REGION Network 72: CM Electrode Cutter Z Axis Command homing
   RUNG wire#powerrail
      Contact( #TRUE )
      Coil( "Unit1.Em4.ControlNodes".cm.Interlock.electrodeCutter.source.homing )
   END_RUNG
   RUNG wire#powerrail
      I_Contact( "Unit1.Em4.ControlNodes".cutter."step".action[113] )
      Not()
      Contact( "Unit1.Em4.ControlNodes".cm.Interlock.electrodeCutter.source.homing )
      Coil( "Unit1.Em4.ControlNodes".cmElectrodeCutterAxisZ.commands.homing )
   END_RUNG
   // the same network as SCL:
   "Unit1.Em4.ControlNodes".cm.Interlock.electrodeCutter.source.homing := #TRUE;
   "Unit1.Em4.ControlNodes".cmElectrodeCutterAxisZ.commands.homing := NOT (NOT "Unit1.Em4.ControlNodes".cutter."step".action[113]) AND "Unit1.Em4.ControlNodes".cm.Interlock.electrodeCutter.source.homing;
END_REGION

REGION Network 73: CM Electrode Cutter Z Axis Command posRelative
   RUNG wire#powerrail
      Contact( #TRUE )
      Coil( "Unit1.Em4.ControlNodes".cm.Interlock.electrodeCutter.source.posRelative )
   END_RUNG
   RUNG wire#powerrail
      I_Contact( "Unit1.Em4.ControlNodes".cutter."step".action[211] )
      Not()
      Coil( "Unit1.Em4.ControlNodes".cmElectrodeCutterAxisZ.commands.posRelative )
   END_RUNG
   // the same network as SCL:
   "Unit1.Em4.ControlNodes".cm.Interlock.electrodeCutter.source.posRelative := #TRUE;
   "Unit1.Em4.ControlNodes".cmElectrodeCutterAxisZ.commands.posRelative := NOT (NOT "Unit1.Em4.ControlNodes".cutter."step".action[211]);
END_REGION

REGION Network 74: CM Electrode Cutter Z Axis Command posAbsolute
   RUNG wire#powerrail
      Contact( #TRUE )
      Coil( "Unit1.Em4.ControlNodes".cm.Interlock.electrodeCutter.source.posAbsolute[0] )
   END_RUNG
   RUNG wire#powerrail
      I_Contact( "Unit1.Em4.ControlNodes".cutter."step".action[122] )
      Not()
      Coil( "Unit1.Em4.ControlNodes".cmElectrodeCutterAxisZ.commands.posAbsolute )
   END_RUNG
   // the same network as SCL:
   "Unit1.Em4.ControlNodes".cm.Interlock.electrodeCutter.source.posAbsolute[0] := #TRUE;
   "Unit1.Em4.ControlNodes".cmElectrodeCutterAxisZ.commands.posAbsolute := NOT (NOT "Unit1.Em4.ControlNodes".cutter."step".action[122]);
END_REGION

REGION Network 75: CM Electrode Cutter Z Axis Command gearInRelative
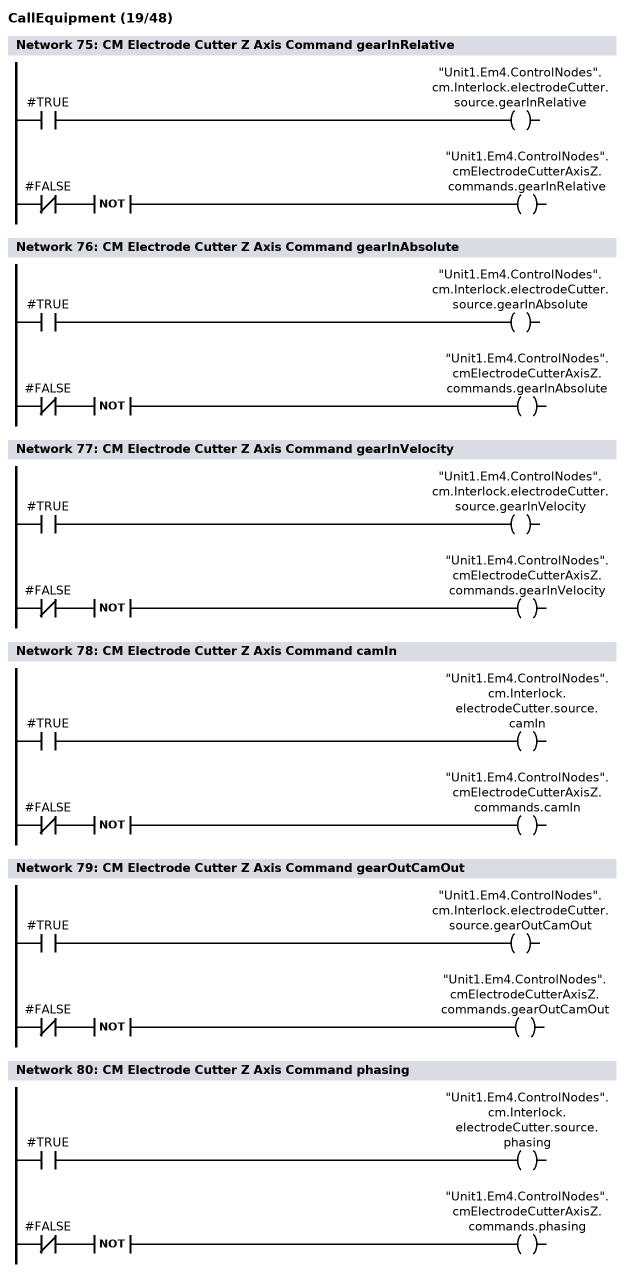
   RUNG wire#powerrail
      Contact( #TRUE )
      Coil( "Unit1.Em4.ControlNodes".cm.Interlock.electrodeCutter.source.gearInRelative )
   END_RUNG
   RUNG wire#powerrail
      I_Contact( #FALSE )
      Not()
      Coil( "Unit1.Em4.ControlNodes".cmElectrodeCutterAxisZ.commands.gearInRelative )
   END_RUNG
   // the same network as SCL:
   "Unit1.Em4.ControlNodes".cm.Interlock.electrodeCutter.source.gearInRelative := #TRUE;
   "Unit1.Em4.ControlNodes".cmElectrodeCutterAxisZ.commands.gearInRelative := NOT (NOT #FALSE);
END_REGION

REGION Network 76: CM Electrode Cutter Z Axis Command gearInAbsolute
   RUNG wire#powerrail
      Contact( #TRUE )
      Coil( "Unit1.Em4.ControlNodes".cm.Interlock.electrodeCutter.source.gearInAbsolute )
   END_RUNG
   RUNG wire#powerrail
      I_Contact( #FALSE )
      Not()
      Coil( "Unit1.Em4.ControlNodes".cmElectrodeCutterAxisZ.commands.gearInAbsolute )
   END_RUNG
   // the same network as SCL:
   "Unit1.Em4.ControlNodes".cm.Interlock.electrodeCutter.source.gearInAbsolute := #TRUE;
   "Unit1.Em4.ControlNodes".cmElectrodeCutterAxisZ.commands.gearInAbsolute := NOT (NOT #FALSE);
END_REGION

REGION Network 77: CM Electrode Cutter Z Axis Command gearInVelocity
   RUNG wire#powerrail
      Contact( #TRUE )
      Coil( "Unit1.Em4.ControlNodes".cm.Interlock.electrodeCutter.source.gearInVelocity )
   END_RUNG
   RUNG wire#powerrail
      I_Contact( #FALSE )
      Not()
      Coil( "Unit1.Em4.ControlNodes".cmElectrodeCutterAxisZ.commands.gearInVelocity )
   END_RUNG
   // the same network as SCL:
   "Unit1.Em4.ControlNodes".cm.Interlock.electrodeCutter.source.gearInVelocity := #TRUE;
   "Unit1.Em4.ControlNodes".cmElectrodeCutterAxisZ.commands.gearInVelocity := NOT (NOT #FALSE);
END_REGION

REGION Network 78: CM Electrode Cutter Z Axis Command camIn
   RUNG wire#powerrail
      Contact( #TRUE )
      Coil( "Unit1.Em4.ControlNodes".cm.Interlock.electrodeCutter.source.camIn )
   END_RUNG
   RUNG wire#powerrail
      I_Contact( #FALSE )
      Not()
      Coil( "Unit1.Em4.ControlNodes".cmElectrodeCutterAxisZ.commands.camIn )
   END_RUNG
   // the same network as SCL:
   "Unit1.Em4.ControlNodes".cm.Interlock.electrodeCutter.source.camIn := #TRUE;
   "Unit1.Em4.ControlNodes".cmElectrodeCutterAxisZ.commands.camIn := NOT (NOT #FALSE);
END_REGION

REGION Network 79: CM Electrode Cutter Z Axis Command gearOutCamOut
   RUNG wire#powerrail
      Contact( #TRUE )
      Coil( "Unit1.Em4.ControlNodes".cm.Interlock.electrodeCutter.source.gearOutCamOut )
   END_RUNG
   RUNG wire#powerrail
      I_Contact( #FALSE )
      Not()
      Coil( "Unit1.Em4.ControlNodes".cmElectrodeCutterAxisZ.commands.gearOutCamOut )
   END_RUNG
   // the same network as SCL:
   "Unit1.Em4.ControlNodes".cm.Interlock.electrodeCutter.source.gearOutCamOut := #TRUE;
   "Unit1.Em4.ControlNodes".cmElectrodeCutterAxisZ.commands.gearOutCamOut := NOT (NOT #FALSE);
END_REGION

REGION Network 80: CM Electrode Cutter Z Axis Command phasing
   RUNG wire#powerrail
      Contact( #TRUE )
      Coil( "Unit1.Em4.ControlNodes".cm.Interlock.electrodeCutter.source.phasing )
   END_RUNG
   RUNG wire#powerrail
      I_Contact( #FALSE )
      Not()
      Coil( "Unit1.Em4.ControlNodes".cmElectrodeCutterAxisZ.commands.phasing )
   END_RUNG
   // the same network as SCL:
   "Unit1.Em4.ControlNodes".cm.Interlock.electrodeCutter.source.phasing := #TRUE;
   "Unit1.Em4.ControlNodes".cmElectrodeCutterAxisZ.commands.phasing := NOT (NOT #FALSE);
END_REGION

REGION Network 81: CM Electrode Cutter Z Axis Command offset
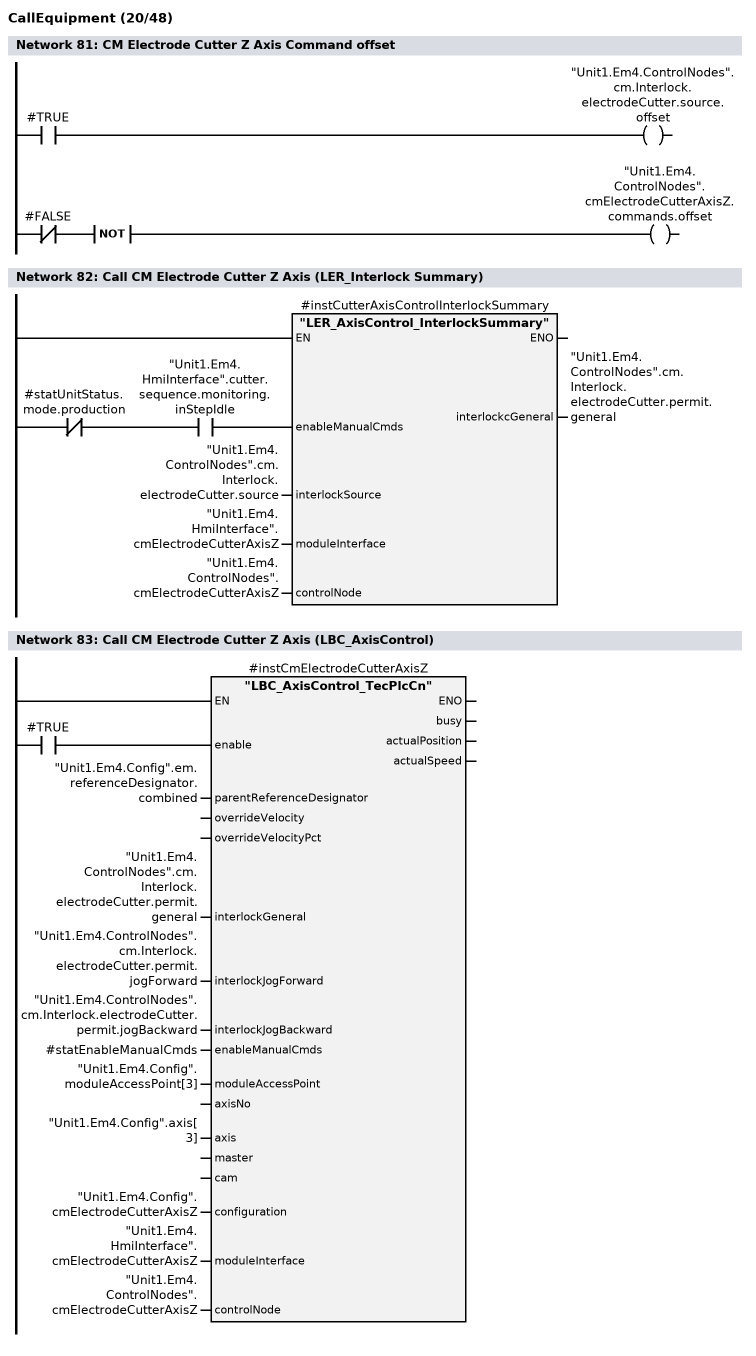
   RUNG wire#powerrail
      Contact( #TRUE )
      Coil( "Unit1.Em4.ControlNodes".cm.Interlock.electrodeCutter.source.offset )
   END_RUNG
   RUNG wire#powerrail
      I_Contact( #FALSE )
      Not()
      Coil( "Unit1.Em4.ControlNodes".cmElectrodeCutterAxisZ.commands.offset )
   END_RUNG
   // the same network as SCL:
   "Unit1.Em4.ControlNodes".cm.Interlock.electrodeCutter.source.offset := #TRUE;
   "Unit1.Em4.ControlNodes".cmElectrodeCutterAxisZ.commands.offset := NOT (NOT #FALSE);
END_REGION

REGION Network 82: Call CM Electrode Cutter Z Axis (LER_Interlock Summary)
   RUNG wire#powerrail
      #instCutterAxisControlInterlockSummary(enableManualCmds := wire#w1, interlockSource := "Unit1.Em4.ControlNodes".cm.Interlock.electrodeCutter.source, moduleInterface := "Unit1.Em4.HmiInterface".cmElectrodeCutterAxisZ, controlNode := "Unit1.Em4.ControlNodes".cmElectrodeCutterAxisZ, interlockcGeneral => "Unit1.Em4.ControlNodes".cm.Interlock.electrodeCutter.permit.general)
   END_RUNG
   RUNG wire#powerrail
      I_Contact( #statUnitStatus.mode.production )
      Contact( "Unit1.Em4.HmiInterface".cutter.sequence.monitoring.inStepIdle )
   END_RUNG wire#w1
   // the same network as SCL:
   #instCutterAxisControlInterlockSummary(enableManualCmds := NOT #statUnitStatus.mode.production AND "Unit1.Em4.HmiInterface".cutter.sequence.monitoring.inStepIdle,   // "LER_AxisControl_InterlockSummary"
                           interlockSource := "Unit1.Em4.ControlNodes".cm.Interlock.electrodeCutter.source,
                           moduleInterface := "Unit1.Em4.HmiInterface".cmElectrodeCutterAxisZ,
                           controlNode := "Unit1.Em4.ControlNodes".cmElectrodeCutterAxisZ,
                           interlockcGeneral => "Unit1.Em4.ControlNodes".cm.Interlock.electrodeCutter.permit.general);
END_REGION

REGION Network 83: Call CM Electrode Cutter Z Axis (LBC_AxisControl)
   RUNG wire#powerrail
      #instCmElectrodeCutterAxisZ(enable := wire#w1, parentReferenceDesignator := "Unit1.Em4.Config".em.referenceDesignator.combined, overrideVelocity :=, overrideVelocityPct :=, interlockGeneral := "Unit1.Em4.ControlNodes".cm.Interlock.electrodeCutter.permit.general, interlockJogForward := "Unit1.Em4.ControlNodes".cm.Interlock.electrodeCutter.permit.jogForward, interlockJogBackward := "Unit1.Em4.ControlNodes".cm.Interlock.electrodeCutter.permit.jogBackward, enableManualCmds := #statEnableManualCmds, moduleAccessPoint := "Unit1.Em4.Config".moduleAccessPoint[3], axisNo :=, axis := "Unit1.Em4.Config".axis[3], master :=, cam :=, configuration := "Unit1.Em4.Config".cmElectrodeCutterAxisZ, moduleInterface := "Unit1.Em4.HmiInterface".cmElectrodeCutterAxisZ, controlNode := "Unit1.Em4.ControlNodes".cmElectrodeCutterAxisZ, busy =>, actualPosition =>, actualSpeed =>)
   END_RUNG
   RUNG wire#powerrail
      Contact( #TRUE )
   END_RUNG wire#w1
   // the same network as SCL:
   #instCmElectrodeCutterAxisZ(enable := #TRUE,   // "LBC_AxisControl_TecPlcCn"
                           parentReferenceDesignator := "Unit1.Em4.Config".em.referenceDesignator.combined,
                           interlockGeneral := "Unit1.Em4.ControlNodes".cm.Interlock.electrodeCutter.permit.general,
                           interlockJogForward := "Unit1.Em4.ControlNodes".cm.Interlock.electrodeCutter.permit.jogForward,
                           interlockJogBackward := "Unit1.Em4.ControlNodes".cm.Interlock.electrodeCutter.permit.jogBackward,
                           enableManualCmds := #statEnableManualCmds,
                           moduleAccessPoint := "Unit1.Em4.Config".moduleAccessPoint[3],
                           axis := "Unit1.Em4.Config".axis[3],
                           configuration := "Unit1.Em4.Config".cmElectrodeCutterAxisZ,
                           moduleInterface := "Unit1.Em4.HmiInterface".cmElectrodeCutterAxisZ,
                           controlNode := "Unit1.Em4.ControlNodes".cmElectrodeCutterAxisZ);
END_REGION

REGION Network 84: Call CM Electrode Cutter Z Axis (LER_ServoTorqueCal)
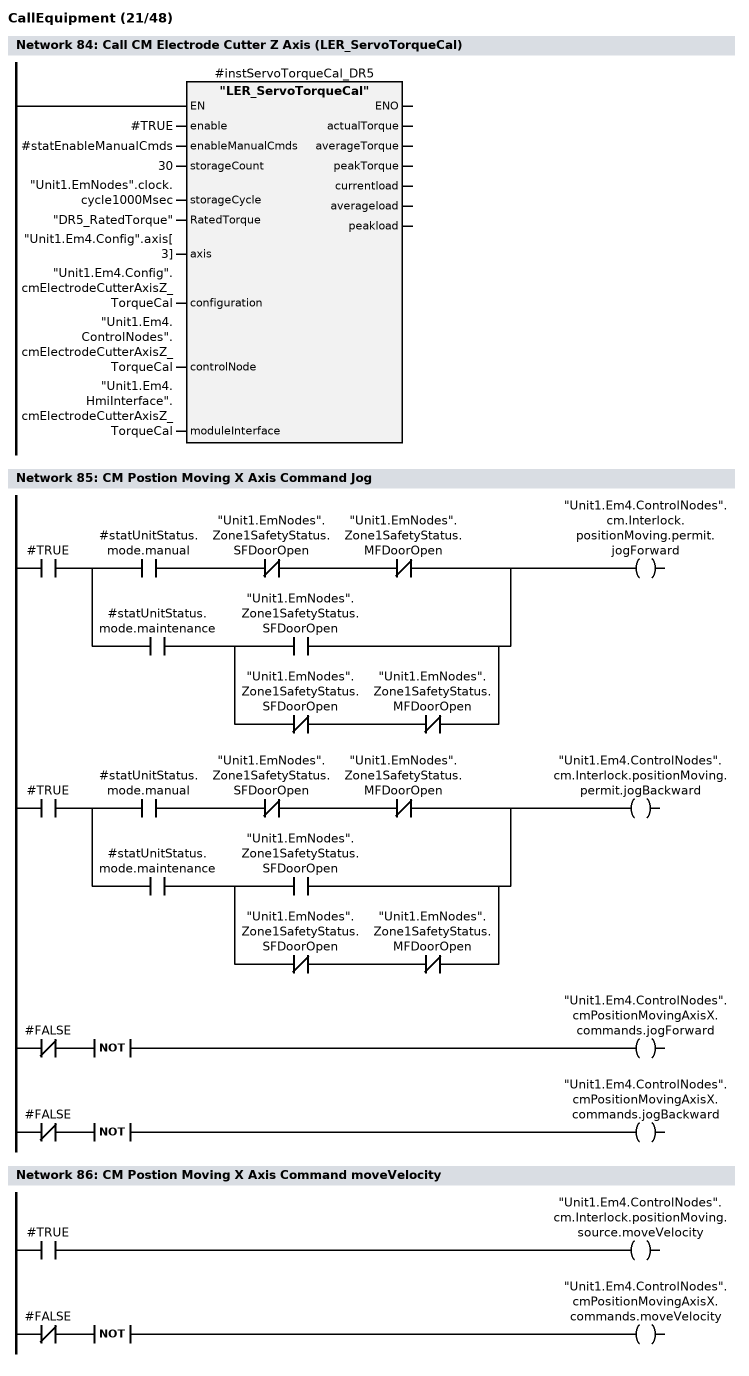
   RUNG wire#powerrail
      #instServoTorqueCal_DR5(enable := #TRUE, enableManualCmds := #statEnableManualCmds, storageCount := 30, storageCycle := "Unit1.EmNodes".clock.cycle1000Msec, RatedTorque := "DR5_RatedTorque", axis := "Unit1.Em4.Config".axis[3], configuration := "Unit1.Em4.Config".cmElectrodeCutterAxisZ_TorqueCal, controlNode := "Unit1.Em4.ControlNodes".cmElectrodeCutterAxisZ_TorqueCal, moduleInterface := "Unit1.Em4.HmiInterface".cmElectrodeCutterAxisZ_TorqueCal, actualTorque =>, averageTorque =>, peakTorque =>, currentload =>, averageload =>, peakload =>)
   END_RUNG
   // the same network as SCL:
   #instServoTorqueCal_DR5(enable := #TRUE,   // "LER_ServoTorqueCal"
                           enableManualCmds := #statEnableManualCmds,
                           storageCount := 30,
                           storageCycle := "Unit1.EmNodes".clock.cycle1000Msec,
                           RatedTorque := "DR5_RatedTorque",
                           axis := "Unit1.Em4.Config".axis[3],
                           configuration := "Unit1.Em4.Config".cmElectrodeCutterAxisZ_TorqueCal,
                           controlNode := "Unit1.Em4.ControlNodes".cmElectrodeCutterAxisZ_TorqueCal,
                           moduleInterface := "Unit1.Em4.HmiInterface".cmElectrodeCutterAxisZ_TorqueCal);
END_REGION

REGION Network 85: CM Postion Moving X Axis Command Jog
   RUNG wire#powerrail
      Contact( #TRUE )
      wire#w1
      Contact( #statUnitStatus.mode.manual )
      I_Contact( "Unit1.EmNodes".Zone1SafetyStatus.SFDoorOpen )
      I_Contact( "Unit1.EmNodes".Zone1SafetyStatus.MFDoorOpen )
      wire#w2
      Coil( "Unit1.Em4.ControlNodes".cm.Interlock.positionMoving.permit.jogForward )
   END_RUNG
   RUNG wire#w1
      Contact( #statUnitStatus.mode.maintenance )
      wire#w3
      Contact( "Unit1.EmNodes".Zone1SafetyStatus.SFDoorOpen )
   END_RUNG wire#w2
   RUNG wire#w3
      I_Contact( "Unit1.EmNodes".Zone1SafetyStatus.SFDoorOpen )
      I_Contact( "Unit1.EmNodes".Zone1SafetyStatus.MFDoorOpen )
   END_RUNG wire#w2
   RUNG wire#powerrail
      Contact( #TRUE )
      wire#w4
      Contact( #statUnitStatus.mode.manual )
      I_Contact( "Unit1.EmNodes".Zone1SafetyStatus.SFDoorOpen )
      I_Contact( "Unit1.EmNodes".Zone1SafetyStatus.MFDoorOpen )
      wire#w5
      Coil( "Unit1.Em4.ControlNodes".cm.Interlock.positionMoving.permit.jogBackward )
   END_RUNG
   RUNG wire#w4
      Contact( #statUnitStatus.mode.maintenance )
      wire#w6
      Contact( "Unit1.EmNodes".Zone1SafetyStatus.SFDoorOpen )
   END_RUNG wire#w5
   RUNG wire#w6
      I_Contact( "Unit1.EmNodes".Zone1SafetyStatus.SFDoorOpen )
      I_Contact( "Unit1.EmNodes".Zone1SafetyStatus.MFDoorOpen )
   END_RUNG wire#w5
   RUNG wire#powerrail
      I_Contact( #FALSE )
      Not()
      Coil( "Unit1.Em4.ControlNodes".cmPositionMovingAxisX.commands.jogForward )
   END_RUNG
   RUNG wire#powerrail
      I_Contact( #FALSE )
      Not()
      Coil( "Unit1.Em4.ControlNodes".cmPositionMovingAxisX.commands.jogBackward )
   END_RUNG
   // the same network as SCL:
   "Unit1.Em4.ControlNodes".cm.Interlock.positionMoving.permit.jogForward := #TRUE AND ((#statUnitStatus.mode.manual AND NOT "Unit1.EmNodes".Zone1SafetyStatus.SFDoorOpen AND NOT "Unit1.EmNodes".Zone1SafetyStatus.MFDoorOpen) OR (#statUnitStatus.mode.maintenance AND ("Unit1.EmNodes".Zone1SafetyStatus.SFDoorOpen OR (NOT "Unit1.EmNodes".Zone1SafetyStatus.SFDoorOpen AND NOT "Unit1.EmNodes".Zone1SafetyStatus.MFDoorOpen))));
   "Unit1.Em4.ControlNodes".cm.Interlock.positionMoving.permit.jogBackward := #TRUE AND ((#statUnitStatus.mode.manual AND NOT "Unit1.EmNodes".Zone1SafetyStatus.SFDoorOpen AND NOT "Unit1.EmNodes".Zone1SafetyStatus.MFDoorOpen) OR (#statUnitStatus.mode.maintenance AND ("Unit1.EmNodes".Zone1SafetyStatus.SFDoorOpen OR (NOT "Unit1.EmNodes".Zone1SafetyStatus.SFDoorOpen AND NOT "Unit1.EmNodes".Zone1SafetyStatus.MFDoorOpen))));
   "Unit1.Em4.ControlNodes".cmPositionMovingAxisX.commands.jogForward := NOT (NOT #FALSE);
   "Unit1.Em4.ControlNodes".cmPositionMovingAxisX.commands.jogBackward := NOT (NOT #FALSE);
END_REGION

REGION Network 86: CM Postion Moving X Axis Command moveVelocity
   RUNG wire#powerrail
      Contact( #TRUE )
      Coil( "Unit1.Em4.ControlNodes".cm.Interlock.positionMoving.source.moveVelocity )
   END_RUNG
   RUNG wire#powerrail
      I_Contact( #FALSE )
      Not()
      Coil( "Unit1.Em4.ControlNodes".cmPositionMovingAxisX.commands.moveVelocity )
   END_RUNG
   // the same network as SCL:
   "Unit1.Em4.ControlNodes".cm.Interlock.positionMoving.source.moveVelocity := #TRUE;
   "Unit1.Em4.ControlNodes".cmPositionMovingAxisX.commands.moveVelocity := NOT (NOT #FALSE);
END_REGION

REGION Network 87: CM Postion Moving X Axis Command stop
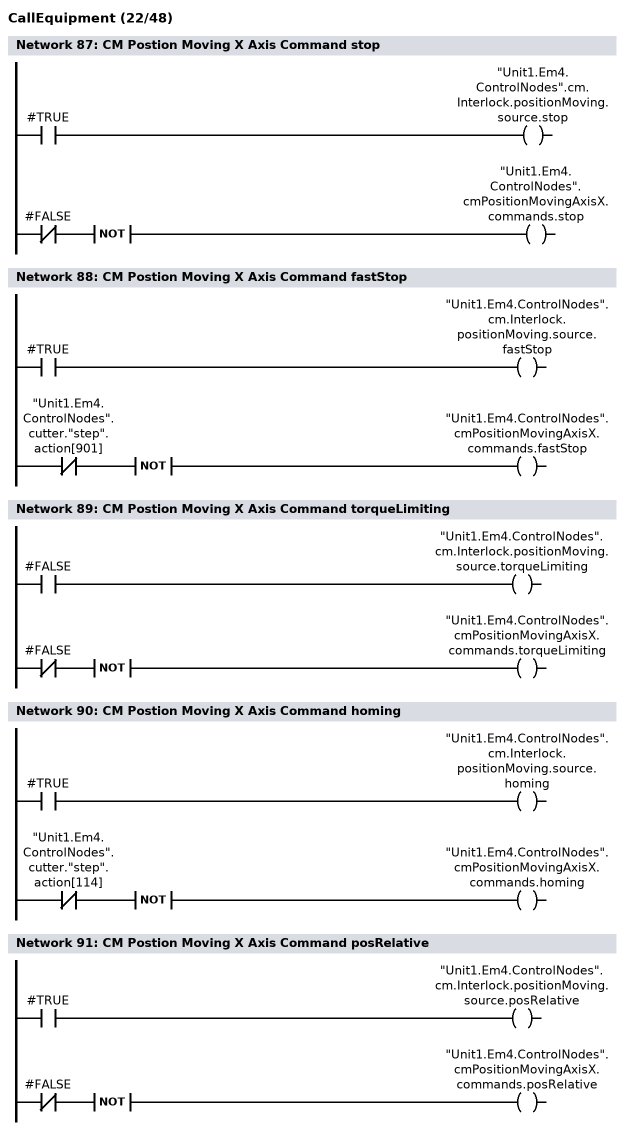
   RUNG wire#powerrail
      Contact( #TRUE )
      Coil( "Unit1.Em4.ControlNodes".cm.Interlock.positionMoving.source.stop )
   END_RUNG
   RUNG wire#powerrail
      I_Contact( #FALSE )
      Not()
      Coil( "Unit1.Em4.ControlNodes".cmPositionMovingAxisX.commands.stop )
   END_RUNG
   // the same network as SCL:
   "Unit1.Em4.ControlNodes".cm.Interlock.positionMoving.source.stop := #TRUE;
   "Unit1.Em4.ControlNodes".cmPositionMovingAxisX.commands.stop := NOT (NOT #FALSE);
END_REGION

REGION Network 88: CM Postion Moving X Axis Command fastStop
   RUNG wire#powerrail
      Contact( #TRUE )
      Coil( "Unit1.Em4.ControlNodes".cm.Interlock.positionMoving.source.fastStop )
   END_RUNG
   RUNG wire#powerrail
      I_Contact( "Unit1.Em4.ControlNodes".cutter."step".action[901] )
      Not()
      Coil( "Unit1.Em4.ControlNodes".cmPositionMovingAxisX.commands.fastStop )
   END_RUNG
   // the same network as SCL:
   "Unit1.Em4.ControlNodes".cm.Interlock.positionMoving.source.fastStop := #TRUE;
   "Unit1.Em4.ControlNodes".cmPositionMovingAxisX.commands.fastStop := NOT (NOT "Unit1.Em4.ControlNodes".cutter."step".action[901]);
END_REGION

REGION Network 89: CM Postion Moving X Axis Command torqueLimiting
   RUNG wire#powerrail
      Contact( #FALSE )
      Coil( "Unit1.Em4.ControlNodes".cm.Interlock.positionMoving.source.torqueLimiting )
   END_RUNG
   RUNG wire#powerrail
      I_Contact( #FALSE )
      Not()
      Coil( "Unit1.Em4.ControlNodes".cmPositionMovingAxisX.commands.torqueLimiting )
   END_RUNG
   // the same network as SCL:
   "Unit1.Em4.ControlNodes".cm.Interlock.positionMoving.source.torqueLimiting := #FALSE;
   "Unit1.Em4.ControlNodes".cmPositionMovingAxisX.commands.torqueLimiting := NOT (NOT #FALSE);
END_REGION

REGION Network 90: CM Postion Moving X Axis Command homing
   RUNG wire#powerrail
      Contact( #TRUE )
      Coil( "Unit1.Em4.ControlNodes".cm.Interlock.positionMoving.source.homing )
   END_RUNG
   RUNG wire#powerrail
      I_Contact( "Unit1.Em4.ControlNodes".cutter."step".action[114] )
      Not()
      Coil( "Unit1.Em4.ControlNodes".cmPositionMovingAxisX.commands.homing )
   END_RUNG
   // the same network as SCL:
   "Unit1.Em4.ControlNodes".cm.Interlock.positionMoving.source.homing := #TRUE;
   "Unit1.Em4.ControlNodes".cmPositionMovingAxisX.commands.homing := NOT (NOT "Unit1.Em4.ControlNodes".cutter."step".action[114]);
END_REGION

REGION Network 91: CM Postion Moving X Axis Command posRelative
   RUNG wire#powerrail
      Contact( #TRUE )
      Coil( "Unit1.Em4.ControlNodes".cm.Interlock.positionMoving.source.posRelative )
   END_RUNG
   RUNG wire#powerrail
      I_Contact( #FALSE )
      Not()
      Coil( "Unit1.Em4.ControlNodes".cmPositionMovingAxisX.commands.posRelative )
   END_RUNG
   // the same network as SCL:
   "Unit1.Em4.ControlNodes".cm.Interlock.positionMoving.source.posRelative := #TRUE;
   "Unit1.Em4.ControlNodes".cmPositionMovingAxisX.commands.posRelative := NOT (NOT #FALSE);
END_REGION

REGION Network 92: CM Postion Moving X Axis Command posAbsolute
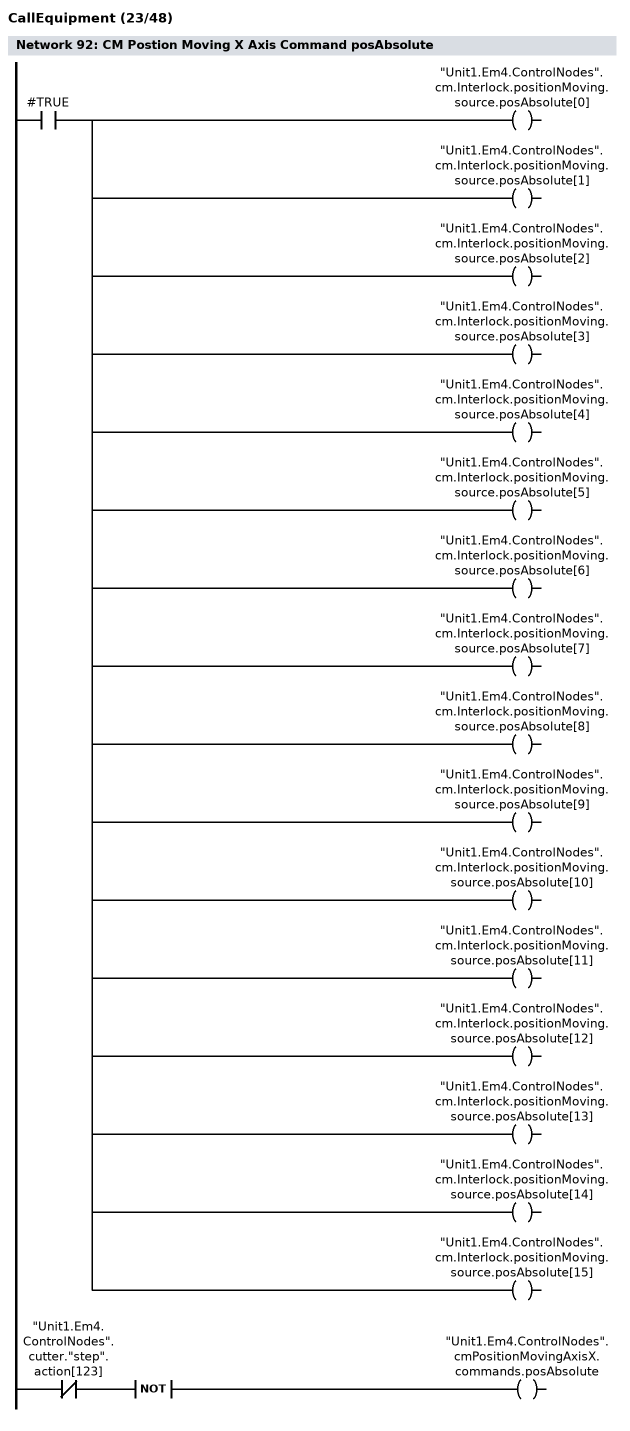
   RUNG wire#powerrail
      Contact( #TRUE )
      wire#w1
      Coil( "Unit1.Em4.ControlNodes".cm.Interlock.positionMoving.source.posAbsolute[0] )
   END_RUNG
   RUNG wire#w1
      Coil( "Unit1.Em4.ControlNodes".cm.Interlock.positionMoving.source.posAbsolute[1] )
   END_RUNG
   RUNG wire#w1
      Coil( "Unit1.Em4.ControlNodes".cm.Interlock.positionMoving.source.posAbsolute[2] )
   END_RUNG
   RUNG wire#w1
      Coil( "Unit1.Em4.ControlNodes".cm.Interlock.positionMoving.source.posAbsolute[3] )
   END_RUNG
   RUNG wire#w1
      Coil( "Unit1.Em4.ControlNodes".cm.Interlock.positionMoving.source.posAbsolute[4] )
   END_RUNG
   RUNG wire#w1
      Coil( "Unit1.Em4.ControlNodes".cm.Interlock.positionMoving.source.posAbsolute[5] )
   END_RUNG
   RUNG wire#w1
      Coil( "Unit1.Em4.ControlNodes".cm.Interlock.positionMoving.source.posAbsolute[6] )
   END_RUNG
   RUNG wire#w1
      Coil( "Unit1.Em4.ControlNodes".cm.Interlock.positionMoving.source.posAbsolute[7] )
   END_RUNG
   RUNG wire#w1
      Coil( "Unit1.Em4.ControlNodes".cm.Interlock.positionMoving.source.posAbsolute[8] )
   END_RUNG
   RUNG wire#w1
      Coil( "Unit1.Em4.ControlNodes".cm.Interlock.positionMoving.source.posAbsolute[9] )
   END_RUNG
   RUNG wire#w1
      Coil( "Unit1.Em4.ControlNodes".cm.Interlock.positionMoving.source.posAbsolute[10] )
   END_RUNG
   RUNG wire#w1
      Coil( "Unit1.Em4.ControlNodes".cm.Interlock.positionMoving.source.posAbsolute[11] )
   END_RUNG
   RUNG wire#w1
      Coil( "Unit1.Em4.ControlNodes".cm.Interlock.positionMoving.source.posAbsolute[12] )
   END_RUNG
   RUNG wire#w1
      Coil( "Unit1.Em4.ControlNodes".cm.Interlock.positionMoving.source.posAbsolute[13] )
   END_RUNG
   RUNG wire#w1
      Coil( "Unit1.Em4.ControlNodes".cm.Interlock.positionMoving.source.posAbsolute[14] )
   END_RUNG
   RUNG wire#w1
      Coil( "Unit1.Em4.ControlNodes".cm.Interlock.positionMoving.source.posAbsolute[15] )
   END_RUNG
   RUNG wire#powerrail
      I_Contact( "Unit1.Em4.ControlNodes".cutter."step".action[123] )
      Not()
      Coil( "Unit1.Em4.ControlNodes".cmPositionMovingAxisX.commands.posAbsolute )
   END_RUNG
   // the same network as SCL:
   "Unit1.Em4.ControlNodes".cm.Interlock.positionMoving.source.posAbsolute[0] := #TRUE;
   "Unit1.Em4.ControlNodes".cm.Interlock.positionMoving.source.posAbsolute[1] := #TRUE;
   "Unit1.Em4.ControlNodes".cm.Interlock.positionMoving.source.posAbsolute[2] := #TRUE;
   "Unit1.Em4.ControlNodes".cm.Interlock.positionMoving.source.posAbsolute[3] := #TRUE;
   "Unit1.Em4.ControlNodes".cm.Interlock.positionMoving.source.posAbsolute[4] := #TRUE;
   "Unit1.Em4.ControlNodes".cm.Interlock.positionMoving.source.posAbsolute[5] := #TRUE;
   "Unit1.Em4.ControlNodes".cm.Interlock.positionMoving.source.posAbsolute[6] := #TRUE;
   "Unit1.Em4.ControlNodes".cm.Interlock.positionMoving.source.posAbsolute[7] := #TRUE;
   "Unit1.Em4.ControlNodes".cm.Interlock.positionMoving.source.posAbsolute[8] := #TRUE;
   "Unit1.Em4.ControlNodes".cm.Interlock.positionMoving.source.posAbsolute[9] := #TRUE;
   "Unit1.Em4.ControlNodes".cm.Interlock.positionMoving.source.posAbsolute[10] := #TRUE;
   "Unit1.Em4.ControlNodes".cm.Interlock.positionMoving.source.posAbsolute[11] := #TRUE;
   "Unit1.Em4.ControlNodes".cm.Interlock.positionMoving.source.posAbsolute[12] := #TRUE;
   "Unit1.Em4.ControlNodes".cm.Interlock.positionMoving.source.posAbsolute[13] := #TRUE;
   "Unit1.Em4.ControlNodes".cm.Interlock.positionMoving.source.posAbsolute[14] := #TRUE;
   "Unit1.Em4.ControlNodes".cm.Interlock.positionMoving.source.posAbsolute[15] := #TRUE;
   "Unit1.Em4.ControlNodes".cmPositionMovingAxisX.commands.posAbsolute := NOT (NOT "Unit1.Em4.ControlNodes".cutter."step".action[123]);
END_REGION

REGION Network 93: Call CM Postion Moving X Axis (LER_Interlock Summary)
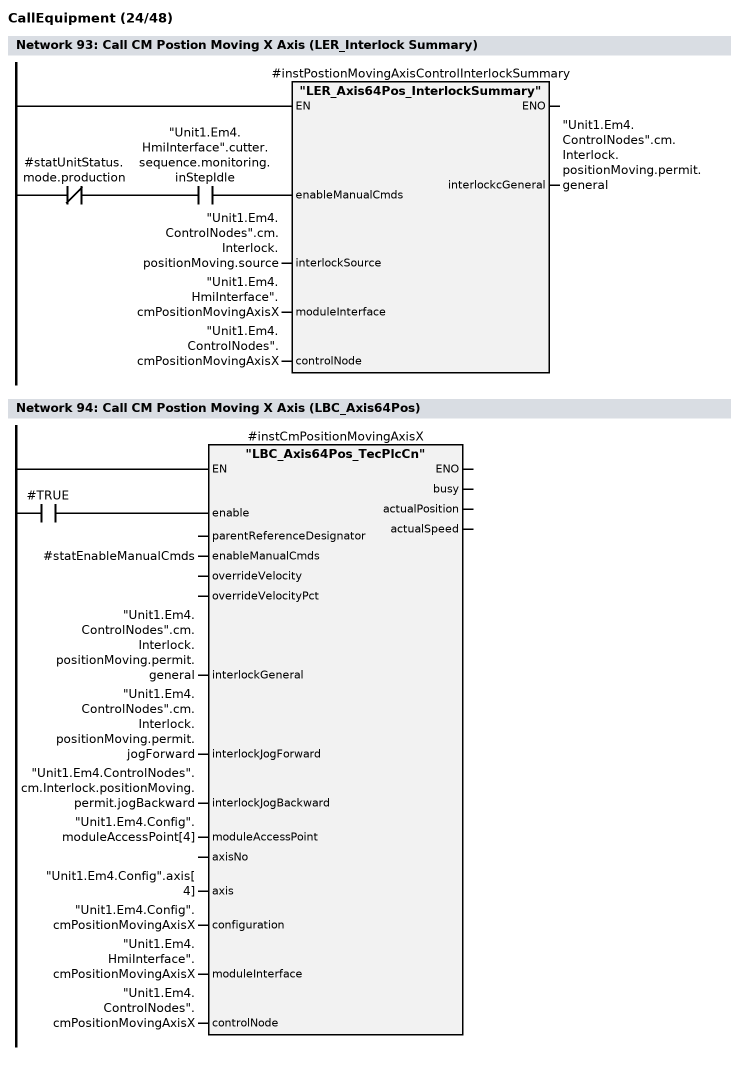
   RUNG wire#powerrail
      #instPostionMovingAxisControlInterlockSummary(enableManualCmds := wire#w1, interlockSource := "Unit1.Em4.ControlNodes".cm.Interlock.positionMoving.source, moduleInterface := "Unit1.Em4.HmiInterface".cmPositionMovingAxisX, controlNode := "Unit1.Em4.ControlNodes".cmPositionMovingAxisX, interlockcGeneral => "Unit1.Em4.ControlNodes".cm.Interlock.positionMoving.permit.general)
   END_RUNG
   RUNG wire#powerrail
      I_Contact( #statUnitStatus.mode.production )
      Contact( "Unit1.Em4.HmiInterface".cutter.sequence.monitoring.inStepIdle )
   END_RUNG wire#w1
   // the same network as SCL:
   #instPostionMovingAxisControlInterlockSummary(enableManualCmds := NOT #statUnitStatus.mode.production AND "Unit1.Em4.HmiInterface".cutter.sequence.monitoring.inStepIdle,   // "LER_Axis64Pos_InterlockSummary"
                           interlockSource := "Unit1.Em4.ControlNodes".cm.Interlock.positionMoving.source,
                           moduleInterface := "Unit1.Em4.HmiInterface".cmPositionMovingAxisX,
                           controlNode := "Unit1.Em4.ControlNodes".cmPositionMovingAxisX,
                           interlockcGeneral => "Unit1.Em4.ControlNodes".cm.Interlock.positionMoving.permit.general);
END_REGION

REGION Network 94: Call CM Postion Moving X Axis (LBC_Axis64Pos)
   RUNG wire#powerrail
      #instCmPositionMovingAxisX(enable := wire#w1, parentReferenceDesignator :=, enableManualCmds := #statEnableManualCmds, overrideVelocity :=, overrideVelocityPct :=, interlockGeneral := "Unit1.Em4.ControlNodes".cm.Interlock.positionMoving.permit.general, interlockJogForward := "Unit1.Em4.ControlNodes".cm.Interlock.positionMoving.permit.jogForward, interlockJogBackward := "Unit1.Em4.ControlNodes".cm.Interlock.positionMoving.permit.jogBackward, moduleAccessPoint := "Unit1.Em4.Config".moduleAccessPoint[4], axisNo :=, axis := "Unit1.Em4.Config".axis[4], configuration := "Unit1.Em4.Config".cmPositionMovingAxisX, moduleInterface := "Unit1.Em4.HmiInterface".cmPositionMovingAxisX, controlNode := "Unit1.Em4.ControlNodes".cmPositionMovingAxisX, busy =>, actualPosition =>, actualSpeed =>)
   END_RUNG
   RUNG wire#powerrail
      Contact( #TRUE )
   END_RUNG wire#w1
   // the same network as SCL:
   #instCmPositionMovingAxisX(enable := #TRUE,   // "LBC_Axis64Pos_TecPlcCn"
                           enableManualCmds := #statEnableManualCmds,
                           interlockGeneral := "Unit1.Em4.ControlNodes".cm.Interlock.positionMoving.permit.general,
                           interlockJogForward := "Unit1.Em4.ControlNodes".cm.Interlock.positionMoving.permit.jogForward,
                           interlockJogBackward := "Unit1.Em4.ControlNodes".cm.Interlock.positionMoving.permit.jogBackward,
                           moduleAccessPoint := "Unit1.Em4.Config".moduleAccessPoint[4],
                           axis := "Unit1.Em4.Config".axis[4],
                           configuration := "Unit1.Em4.Config".cmPositionMovingAxisX,
                           moduleInterface := "Unit1.Em4.HmiInterface".cmPositionMovingAxisX,
                           controlNode := "Unit1.Em4.ControlNodes".cmPositionMovingAxisX);
END_REGION

REGION Network 95: Call CM Postion Moving X Axis (LER_ServoTorqueCal)
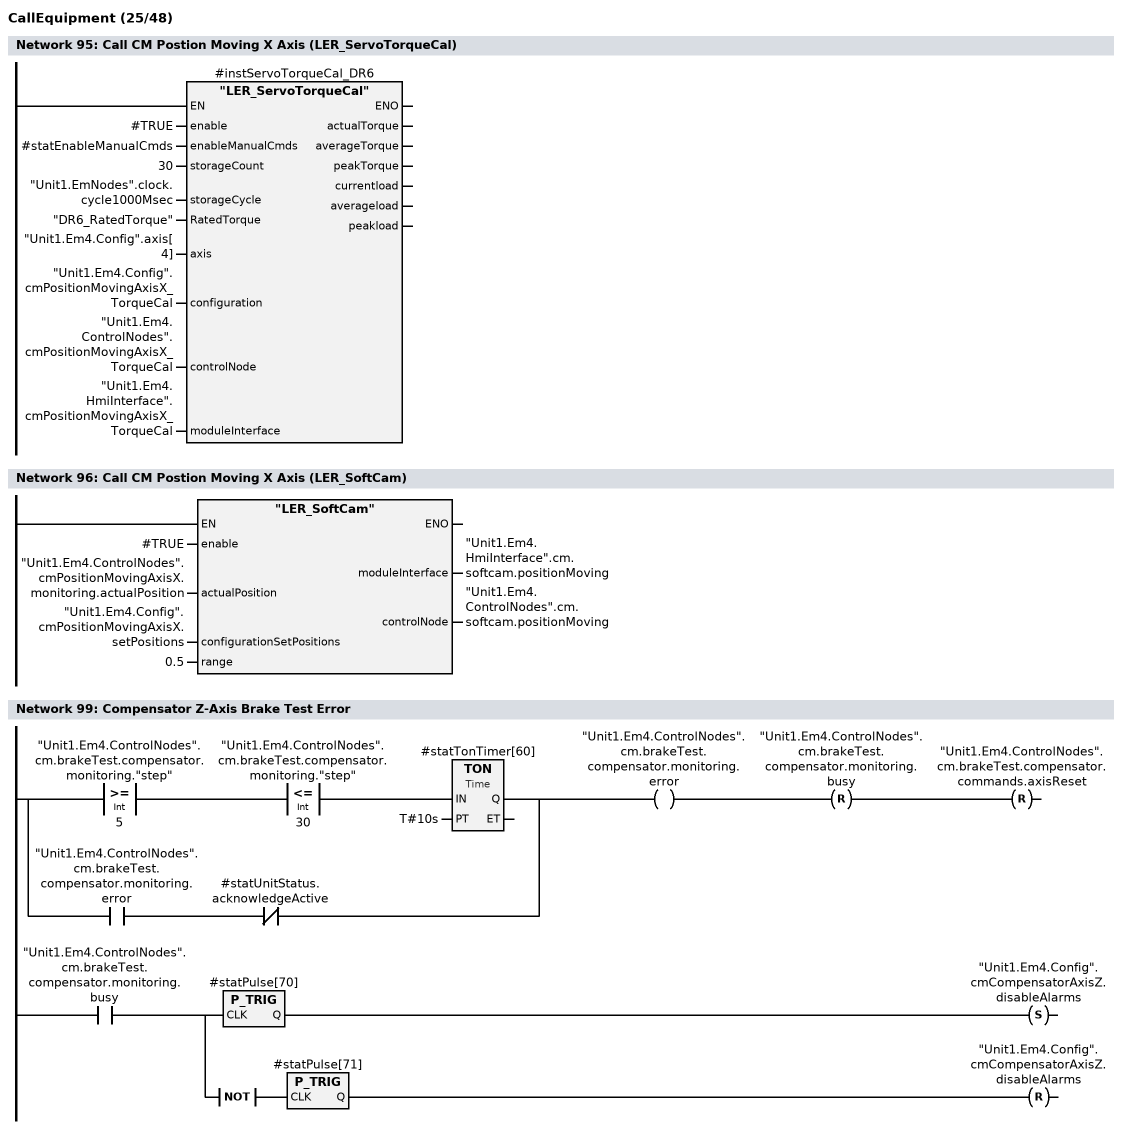
   RUNG wire#powerrail
      #instServoTorqueCal_DR6(enable := #TRUE, enableManualCmds := #statEnableManualCmds, storageCount := 30, storageCycle := "Unit1.EmNodes".clock.cycle1000Msec, RatedTorque := "DR6_RatedTorque", axis := "Unit1.Em4.Config".axis[4], configuration := "Unit1.Em4.Config".cmPositionMovingAxisX_TorqueCal, controlNode := "Unit1.Em4.ControlNodes".cmPositionMovingAxisX_TorqueCal, moduleInterface := "Unit1.Em4.HmiInterface".cmPositionMovingAxisX_TorqueCal, actualTorque =>, averageTorque =>, peakTorque =>, currentload =>, averageload =>, peakload =>)
   END_RUNG
   // the same network as SCL:
   #instServoTorqueCal_DR6(enable := #TRUE,   // "LER_ServoTorqueCal"
                           enableManualCmds := #statEnableManualCmds,
                           storageCount := 30,
                           storageCycle := "Unit1.EmNodes".clock.cycle1000Msec,
                           RatedTorque := "DR6_RatedTorque",
                           axis := "Unit1.Em4.Config".axis[4],
                           configuration := "Unit1.Em4.Config".cmPositionMovingAxisX_TorqueCal,
                           controlNode := "Unit1.Em4.ControlNodes".cmPositionMovingAxisX_TorqueCal,
                           moduleInterface := "Unit1.Em4.HmiInterface".cmPositionMovingAxisX_TorqueCal);
END_REGION

REGION Network 96: Call CM Postion Moving X Axis (LER_SoftCam)
   RUNG wire#powerrail
      "LER_SoftCam"(enable := #TRUE, actualPosition := "Unit1.Em4.ControlNodes".cmPositionMovingAxisX.monitoring.actualPosition, configurationSetPositions := "Unit1.Em4.Config".cmPositionMovingAxisX.setPositions, range := 0.5, moduleInterface => "Unit1.Em4.HmiInterface".cm.softcam.positionMoving, controlNode => "Unit1.Em4.ControlNodes".cm.softcam.positionMoving)
   END_RUNG
   // the same network as SCL:
   "LER_SoftCam"(enable := #TRUE,
                 actualPosition := "Unit1.Em4.ControlNodes".cmPositionMovingAxisX.monitoring.actualPosition,
                 configurationSetPositions := "Unit1.Em4.Config".cmPositionMovingAxisX.setPositions,
                 range := 0.5,
                 moduleInterface => "Unit1.Em4.HmiInterface".cm.softcam.positionMoving,
                 controlNode => "Unit1.Em4.ControlNodes".cm.softcam.positionMoving);
END_REGION

REGION Network 98: ******************** Brake Test (Axis) ********************
END_REGION

REGION Network 99: Compensator Z-Axis Brake Test Error
   RUNG wire#powerrail
      { S7_Templates := "SrcType := Int" } GE_Contact(in1 := "Unit1.Em4.ControlNodes".cm.brakeTest.compensator.monitoring."step", in2 := 5)
      { S7_Templates := "SrcType := Int" } LE_Contact(in1 := "Unit1.Em4.ControlNodes".cm.brakeTest.compensator.monitoring."step", in2 := 30)
      { S7_Templates := "time_type := Time" } #statTonTimer[60].TON(pt := T#10s, et =>)
      wire#w1
      Coil( "Unit1.Em4.ControlNodes".cm.brakeTest.compensator.monitoring.error )
      R_Coil( "Unit1.Em4.ControlNodes".cm.brakeTest.compensator.monitoring.busy )
      R_Coil( "Unit1.Em4.ControlNodes".cm.brakeTest.compensator.commands.axisReset )
   END_RUNG
   RUNG wire#powerrail
      Contact( "Unit1.Em4.ControlNodes".cm.brakeTest.compensator.monitoring.error )
      I_Contact( #statUnitStatus.acknowledgeActive )
   END_RUNG wire#w1
   RUNG wire#powerrail
      Contact( "Unit1.Em4.ControlNodes".cm.brakeTest.compensator.monitoring.busy )
      wire#w2
      P_Trig( #statPulse[70] )
      S_Coil( "Unit1.Em4.Config".cmCompensatorAxisZ.disableAlarms )
   END_RUNG
   RUNG wire#w2
      Not()
      P_Trig( #statPulse[71] )
      R_Coil( "Unit1.Em4.Config".cmCompensatorAxisZ.disableAlarms )
   END_RUNG
   // the same network as SCL:
   #statTonTimer[60].TON(IN := ("Unit1.Em4.ControlNodes".cm.brakeTest.compensator.monitoring."step" >= 5) AND ("Unit1.Em4.ControlNodes".cm.brakeTest.compensator.monitoring."step" <= 30),
                         PT := T#10s);
   "Unit1.Em4.ControlNodes".cm.brakeTest.compensator.monitoring.error := #statTonTimer[60].Q OR ("Unit1.Em4.ControlNodes".cm.brakeTest.compensator.monitoring.error AND NOT #statUnitStatus.acknowledgeActive);
   IF "Unit1.Em4.ControlNodes".cm.brakeTest.compensator.monitoring.error THEN
       "Unit1.Em4.ControlNodes".cm.brakeTest.compensator.monitoring.busy := FALSE;
       "Unit1.Em4.ControlNodes".cm.brakeTest.compensator.commands.axisReset := FALSE;
   END_IF;
   #_w1 := "Unit1.Em4.ControlNodes".cm.brakeTest.compensator.monitoring.busy AND NOT #statPulse[70];   // rising edge
   #statPulse[70] := "Unit1.Em4.ControlNodes".cm.brakeTest.compensator.monitoring.busy;
   IF #_w1 THEN "Unit1.Em4.Config".cmCompensatorAxisZ.disableAlarms := TRUE; END_IF;
   #_w2 := NOT "Unit1.Em4.ControlNodes".cm.brakeTest.compensator.monitoring.busy AND NOT #statPulse[71];   // rising edge
   #statPulse[71] := NOT "Unit1.Em4.ControlNodes".cm.brakeTest.compensator.monitoring.busy;
   IF #_w2 THEN "Unit1.Em4.Config".cmCompensatorAxisZ.disableAlarms := FALSE; END_IF;
END_REGION

REGION Network 100: Compensator Z-Axis Brake Test Initialize
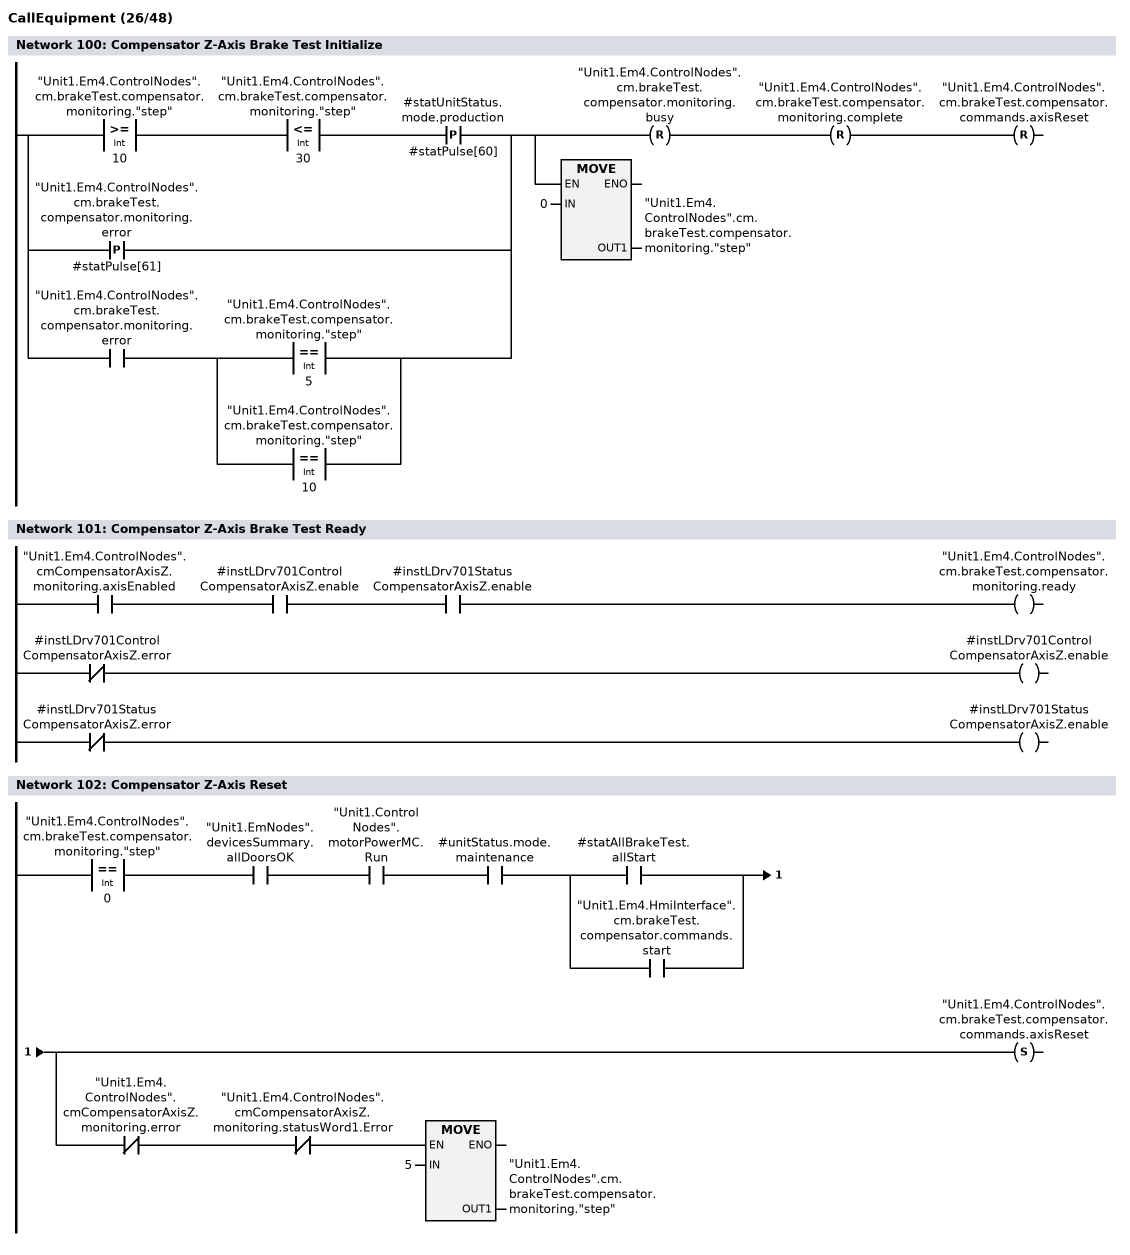
   RUNG wire#powerrail
      { S7_Templates := "SrcType := Int" } GE_Contact(in1 := "Unit1.Em4.ControlNodes".cm.brakeTest.compensator.monitoring."step", in2 := 10)
      { S7_Templates := "SrcType := Int" } LE_Contact(in1 := "Unit1.Em4.ControlNodes".cm.brakeTest.compensator.monitoring."step", in2 := 30)
      P_Contact(operand := #statUnitStatus.mode.production, bit := #statPulse[60])
      wire#w1
      R_Coil( "Unit1.Em4.ControlNodes".cm.brakeTest.compensator.monitoring.busy )
      R_Coil( "Unit1.Em4.ControlNodes".cm.brakeTest.compensator.monitoring.complete )
      R_Coil( "Unit1.Em4.ControlNodes".cm.brakeTest.compensator.commands.axisReset )
   END_RUNG
   RUNG wire#powerrail
      P_Contact(operand := "Unit1.Em4.ControlNodes".cm.brakeTest.compensator.monitoring.error, bit := #statPulse[61])
   END_RUNG wire#w1
   RUNG wire#powerrail
      Contact( "Unit1.Em4.ControlNodes".cm.brakeTest.compensator.monitoring.error )
      wire#w2
      { S7_Templates := "SrcType := Int" } EQ_Contact(in1 := "Unit1.Em4.ControlNodes".cm.brakeTest.compensator.monitoring."step", in2 := 5)
   END_RUNG wire#w1
   RUNG wire#w2
      { S7_Templates := "SrcType := Int" } EQ_Contact(in1 := "Unit1.Em4.ControlNodes".cm.brakeTest.compensator.monitoring."step", in2 := 10)
   END_RUNG wire#w1
   RUNG wire#w1
      Move(in := 0, out1 => "Unit1.Em4.ControlNodes".cm.brakeTest.compensator.monitoring."step")
   END_RUNG
   // the same network as SCL:
   #_w1 := ("Unit1.Em4.ControlNodes".cm.brakeTest.compensator.monitoring."step" >= 10) AND ("Unit1.Em4.ControlNodes".cm.brakeTest.compensator.monitoring."step" <= 30) AND #statUnitStatus.mode.production AND NOT #statPulse[60];   // rising edge of #statUnitStatus.mode.production
   #statPulse[60] := #statUnitStatus.mode.production;
   #_w2 := "Unit1.Em4.ControlNodes".cm.brakeTest.compensator.monitoring.error AND NOT #statPulse[61];   // rising edge of "Unit1.Em4.ControlNodes".cm.brakeTest.compensator.monitoring.error
   #statPulse[61] := "Unit1.Em4.ControlNodes".cm.brakeTest.compensator.monitoring.error;
   IF #_w1 OR #_w2 OR ("Unit1.Em4.ControlNodes".cm.brakeTest.compensator.monitoring.error AND (("Unit1.Em4.ControlNodes".cm.brakeTest.compensator.monitoring."step" = 5) OR ("Unit1.Em4.ControlNodes".cm.brakeTest.compensator.monitoring."step" = 10))) THEN
       "Unit1.Em4.ControlNodes".cm.brakeTest.compensator.monitoring.busy := FALSE;
       "Unit1.Em4.ControlNodes".cm.brakeTest.compensator.monitoring.complete := FALSE;
       "Unit1.Em4.ControlNodes".cm.brakeTest.compensator.commands.axisReset := FALSE;
       "Unit1.Em4.ControlNodes".cm.brakeTest.compensator.monitoring."step" := 0;
   END_IF;
END_REGION

REGION Network 101: Compensator Z-Axis Brake Test Ready
   RUNG wire#powerrail
      Contact( "Unit1.Em4.ControlNodes".cmCompensatorAxisZ.monitoring.axisEnabled )
      Contact( #instLDrv701ControlCompensatorAxisZ.enable )
      Contact( #instLDrv701StatusCompensatorAxisZ.enable )
      Coil( "Unit1.Em4.ControlNodes".cm.brakeTest.compensator.monitoring.ready )
   END_RUNG
   RUNG wire#powerrail
      I_Contact( #instLDrv701ControlCompensatorAxisZ.error )
      Coil( #instLDrv701ControlCompensatorAxisZ.enable )
   END_RUNG
   RUNG wire#powerrail
      I_Contact( #instLDrv701StatusCompensatorAxisZ.error )
      Coil( #instLDrv701StatusCompensatorAxisZ.enable )
   END_RUNG
   // the same network as SCL:
   "Unit1.Em4.ControlNodes".cm.brakeTest.compensator.monitoring.ready := "Unit1.Em4.ControlNodes".cmCompensatorAxisZ.monitoring.axisEnabled AND #instLDrv701ControlCompensatorAxisZ.enable AND #instLDrv701StatusCompensatorAxisZ.enable;
   #instLDrv701ControlCompensatorAxisZ.enable := NOT #instLDrv701ControlCompensatorAxisZ.error;
   #instLDrv701StatusCompensatorAxisZ.enable := NOT #instLDrv701StatusCompensatorAxisZ.error;
END_REGION

REGION Network 102: Compensator Z-Axis Reset
   RUNG wire#powerrail
      { S7_Templates := "SrcType := Int" } EQ_Contact(in1 := "Unit1.Em4.ControlNodes".cm.brakeTest.compensator.monitoring."step", in2 := 0)
      Contact( "Unit1.EmNodes".devicesSummary.allDoorsOK )
      Contact( "Unit1.ControlNodes".motorPowerMC.Run )
      Contact( #unitStatus.mode.maintenance )
      wire#w1
      Contact( #statAllBrakeTest.allStart )
      wire#w2
      S_Coil( "Unit1.Em4.ControlNodes".cm.brakeTest.compensator.commands.axisReset )
   END_RUNG
   RUNG wire#w1
      Contact( "Unit1.Em4.HmiInterface".cm.brakeTest.compensator.commands.start )
   END_RUNG wire#w2
   RUNG wire#w2
      I_Contact( "Unit1.Em4.ControlNodes".cmCompensatorAxisZ.monitoring.error )
      I_Contact( "Unit1.Em4.ControlNodes".cmCompensatorAxisZ.monitoring.statusWord1.Error )
      Move(in := 5, out1 => "Unit1.Em4.ControlNodes".cm.brakeTest.compensator.monitoring."step")
   END_RUNG
   // the same network as SCL:
   #_w1 := ("Unit1.Em4.ControlNodes".cm.brakeTest.compensator.monitoring."step" = 0) AND "Unit1.EmNodes".devicesSummary.allDoorsOK AND "Unit1.ControlNodes".motorPowerMC.Run AND #unitStatus.mode.maintenance AND (#statAllBrakeTest.allStart OR "Unit1.Em4.HmiInterface".cm.brakeTest.compensator.commands.start);
   IF #_w1 THEN "Unit1.Em4.ControlNodes".cm.brakeTest.compensator.commands.axisReset := TRUE; END_IF;
   IF #_w1 AND NOT "Unit1.Em4.ControlNodes".cmCompensatorAxisZ.monitoring.error AND NOT "Unit1.Em4.ControlNodes".cmCompensatorAxisZ.monitoring.statusWord1.Error THEN
       "Unit1.Em4.ControlNodes".cm.brakeTest.compensator.monitoring."step" := 5;
   END_IF;
END_REGION

REGION Network 103: Compensator Z-Axis Brake Test Commands
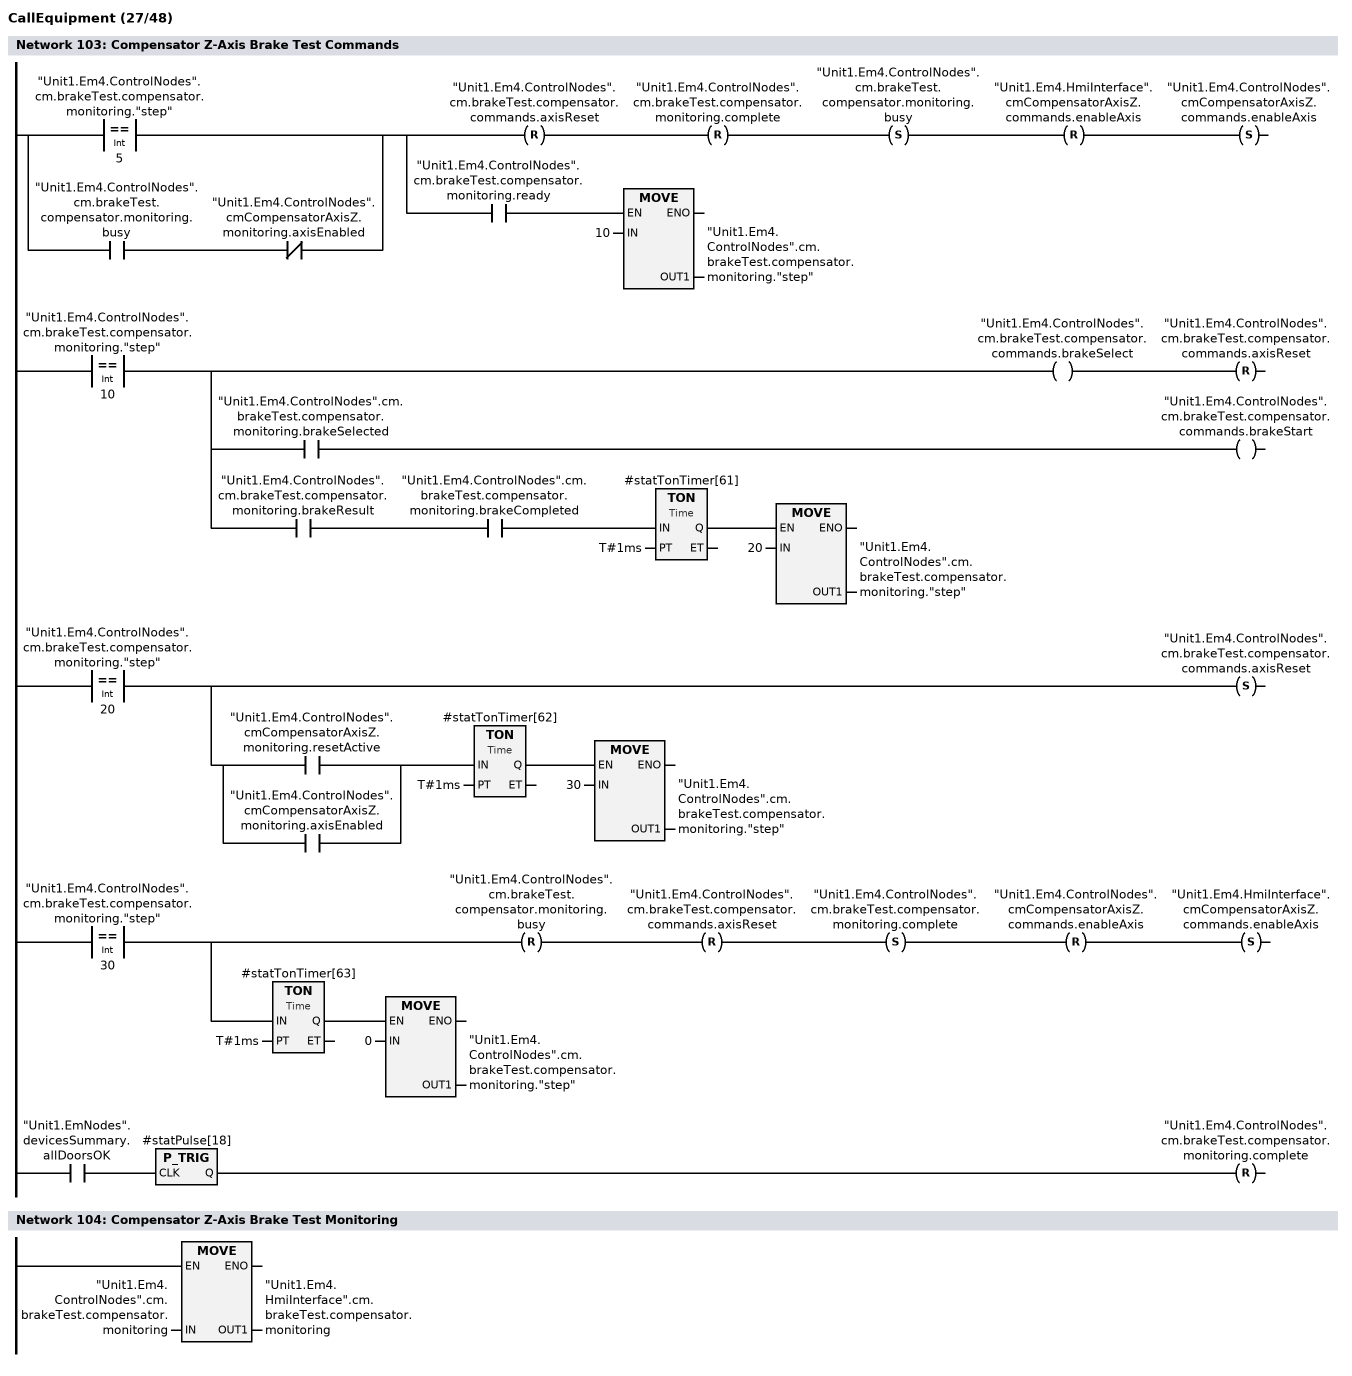
   RUNG wire#powerrail
      { S7_Templates := "SrcType := Int" } EQ_Contact(in1 := "Unit1.Em4.ControlNodes".cm.brakeTest.compensator.monitoring."step", in2 := 5)
      wire#w1
      R_Coil( "Unit1.Em4.ControlNodes".cm.brakeTest.compensator.commands.axisReset )
      R_Coil( "Unit1.Em4.ControlNodes".cm.brakeTest.compensator.monitoring.complete )
      S_Coil( "Unit1.Em4.ControlNodes".cm.brakeTest.compensator.monitoring.busy )
      R_Coil( "Unit1.Em4.HmiInterface".cmCompensatorAxisZ.commands.enableAxis )
      S_Coil( "Unit1.Em4.ControlNodes".cmCompensatorAxisZ.commands.enableAxis )
   END_RUNG
   RUNG wire#powerrail
      Contact( "Unit1.Em4.ControlNodes".cm.brakeTest.compensator.monitoring.busy )
      I_Contact( "Unit1.Em4.ControlNodes".cmCompensatorAxisZ.monitoring.axisEnabled )
   END_RUNG wire#w1
   RUNG wire#w1
      Contact( "Unit1.Em4.ControlNodes".cm.brakeTest.compensator.monitoring.ready )
      Move(in := 10, out1 => "Unit1.Em4.ControlNodes".cm.brakeTest.compensator.monitoring."step")
   END_RUNG
   RUNG wire#powerrail
      { S7_Templates := "SrcType := Int" } EQ_Contact(in1 := "Unit1.Em4.ControlNodes".cm.brakeTest.compensator.monitoring."step", in2 := 10)
      wire#w2
      Coil( "Unit1.Em4.ControlNodes".cm.brakeTest.compensator.commands.brakeSelect )
      R_Coil( "Unit1.Em4.ControlNodes".cm.brakeTest.compensator.commands.axisReset )
   END_RUNG
   RUNG wire#w2
      Contact( "Unit1.Em4.ControlNodes".cm.brakeTest.compensator.monitoring.brakeSelected )
      Coil( "Unit1.Em4.ControlNodes".cm.brakeTest.compensator.commands.brakeStart )
   END_RUNG
   RUNG wire#w2
      Contact( "Unit1.Em4.ControlNodes".cm.brakeTest.compensator.monitoring.brakeResult )
      Contact( "Unit1.Em4.ControlNodes".cm.brakeTest.compensator.monitoring.brakeCompleted )
      { S7_Templates := "time_type := Time" } #statTonTimer[61].TON(pt := T#1ms, et =>)
      Move(in := 20, out1 => "Unit1.Em4.ControlNodes".cm.brakeTest.compensator.monitoring."step")
   END_RUNG
   RUNG wire#powerrail
      { S7_Templates := "SrcType := Int" } EQ_Contact(in1 := "Unit1.Em4.ControlNodes".cm.brakeTest.compensator.monitoring."step", in2 := 20)
      wire#w3
      S_Coil( "Unit1.Em4.ControlNodes".cm.brakeTest.compensator.commands.axisReset )
   END_RUNG
   RUNG wire#w3
      Contact( "Unit1.Em4.ControlNodes".cmCompensatorAxisZ.monitoring.resetActive )
      wire#w4
      { S7_Templates := "time_type := Time" } #statTonTimer[62].TON(pt := T#1ms, et =>)
      Move(in := 30, out1 => "Unit1.Em4.ControlNodes".cm.brakeTest.compensator.monitoring."step")
   END_RUNG
   RUNG wire#w3
      Contact( "Unit1.Em4.ControlNodes".cmCompensatorAxisZ.monitoring.axisEnabled )
   END_RUNG wire#w4
   RUNG wire#powerrail
      { S7_Templates := "SrcType := Int" } EQ_Contact(in1 := "Unit1.Em4.ControlNodes".cm.brakeTest.compensator.monitoring."step", in2 := 30)
      wire#w5
      R_Coil( "Unit1.Em4.ControlNodes".cm.brakeTest.compensator.monitoring.busy )
      R_Coil( "Unit1.Em4.ControlNodes".cm.brakeTest.compensator.commands.axisReset )
      S_Coil( "Unit1.Em4.ControlNodes".cm.brakeTest.compensator.monitoring.complete )
      R_Coil( "Unit1.Em4.ControlNodes".cmCompensatorAxisZ.commands.enableAxis )
      S_Coil( "Unit1.Em4.HmiInterface".cmCompensatorAxisZ.commands.enableAxis )
   END_RUNG
   RUNG wire#w5
      { S7_Templates := "time_type := Time" } #statTonTimer[63].TON(pt := T#1ms, et =>)
      Move(in := 0, out1 => "Unit1.Em4.ControlNodes".cm.brakeTest.compensator.monitoring."step")
   END_RUNG
   RUNG wire#powerrail
      Contact( "Unit1.EmNodes".devicesSummary.allDoorsOK )
      P_Trig( #statPulse[18] )
      R_Coil( "Unit1.Em4.ControlNodes".cm.brakeTest.compensator.monitoring.complete )
   END_RUNG
   // the same network as SCL:
   #_w1 := ("Unit1.Em4.ControlNodes".cm.brakeTest.compensator.monitoring."step" = 5) OR ("Unit1.Em4.ControlNodes".cm.brakeTest.compensator.monitoring.busy AND NOT "Unit1.Em4.ControlNodes".cmCompensatorAxisZ.monitoring.axisEnabled);
   IF #_w1 THEN
       "Unit1.Em4.ControlNodes".cm.brakeTest.compensator.commands.axisReset := FALSE;
       "Unit1.Em4.ControlNodes".cm.brakeTest.compensator.monitoring.complete := FALSE;
       "Unit1.Em4.ControlNodes".cm.brakeTest.compensator.monitoring.busy := TRUE;
       "Unit1.Em4.HmiInterface".cmCompensatorAxisZ.commands.enableAxis := FALSE;
       "Unit1.Em4.ControlNodes".cmCompensatorAxisZ.commands.enableAxis := TRUE;
   END_IF;
   IF #_w1 AND "Unit1.Em4.ControlNodes".cm.brakeTest.compensator.monitoring.ready THEN
       "Unit1.Em4.ControlNodes".cm.brakeTest.compensator.monitoring."step" := 10;
   END_IF;
   "Unit1.Em4.ControlNodes".cm.brakeTest.compensator.commands.brakeSelect := "Unit1.Em4.ControlNodes".cm.brakeTest.compensator.monitoring."step" = 10;
   IF "Unit1.Em4.ControlNodes".cm.brakeTest.compensator.commands.brakeSelect THEN
       "Unit1.Em4.ControlNodes".cm.brakeTest.compensator.commands.axisReset := FALSE;
   END_IF;
   "Unit1.Em4.ControlNodes".cm.brakeTest.compensator.commands.brakeStart := "Unit1.Em4.ControlNodes".cm.brakeTest.compensator.commands.brakeSelect AND "Unit1.Em4.ControlNodes".cm.brakeTest.compensator.monitoring.brakeSelected;
   #statTonTimer[61].TON(IN := "Unit1.Em4.ControlNodes".cm.brakeTest.compensator.commands.brakeSelect AND "Unit1.Em4.ControlNodes".cm.brakeTest.compensator.monitoring.brakeResult AND "Unit1.Em4.ControlNodes".cm.brakeTest.compensator.monitoring.brakeCompleted,
                         PT := T#1ms);
   IF #statTonTimer[61].Q THEN
       "Unit1.Em4.ControlNodes".cm.brakeTest.compensator.monitoring."step" := 20;
   END_IF;
   #_w2 := "Unit1.Em4.ControlNodes".cm.brakeTest.compensator.monitoring."step" = 20;
   IF #_w2 THEN "Unit1.Em4.ControlNodes".cm.brakeTest.compensator.commands.axisReset := TRUE; END_IF;
   #statTonTimer[62].TON(IN := #_w2 AND ("Unit1.Em4.ControlNodes".cmCompensatorAxisZ.monitoring.resetActive OR "Unit1.Em4.ControlNodes".cmCompensatorAxisZ.monitoring.axisEnabled),
                         PT := T#1ms);
   IF #statTonTimer[62].Q THEN
       "Unit1.Em4.ControlNodes".cm.brakeTest.compensator.monitoring."step" := 30;
   END_IF;
   #_w3 := "Unit1.Em4.ControlNodes".cm.brakeTest.compensator.monitoring."step" = 30;
   IF #_w3 THEN
       "Unit1.Em4.ControlNodes".cm.brakeTest.compensator.monitoring.busy := FALSE;
       "Unit1.Em4.ControlNodes".cm.brakeTest.compensator.commands.axisReset := FALSE;
       "Unit1.Em4.ControlNodes".cm.brakeTest.compensator.monitoring.complete := TRUE;
       "Unit1.Em4.ControlNodes".cmCompensatorAxisZ.commands.enableAxis := FALSE;
       "Unit1.Em4.HmiInterface".cmCompensatorAxisZ.commands.enableAxis := TRUE;
   END_IF;
   #statTonTimer[63].TON(IN := #_w3, PT := T#1ms);
   IF #statTonTimer[63].Q THEN
       "Unit1.Em4.ControlNodes".cm.brakeTest.compensator.monitoring."step" := 0;
   END_IF;
   #_w4 := "Unit1.EmNodes".devicesSummary.allDoorsOK AND NOT #statPulse[18];   // rising edge
   #statPulse[18] := "Unit1.EmNodes".devicesSummary.allDoorsOK;
   IF #_w4 THEN "Unit1.Em4.ControlNodes".cm.brakeTest.compensator.monitoring.complete := FALSE; END_IF;
END_REGION

REGION Network 104: Compensator Z-Axis Brake Test Monitoring
   RUNG wire#powerrail
      Move(in := "Unit1.Em4.ControlNodes".cm.brakeTest.compensator.monitoring, out1 => "Unit1.Em4.HmiInterface".cm.brakeTest.compensator.monitoring)
   END_RUNG
   // the same network as SCL:
   "Unit1.Em4.HmiInterface".cm.brakeTest.compensator.monitoring := "Unit1.Em4.ControlNodes".cm.brakeTest.compensator.monitoring;
END_REGION

REGION Network 105: Call Compensator Z-Axis Telegram 701
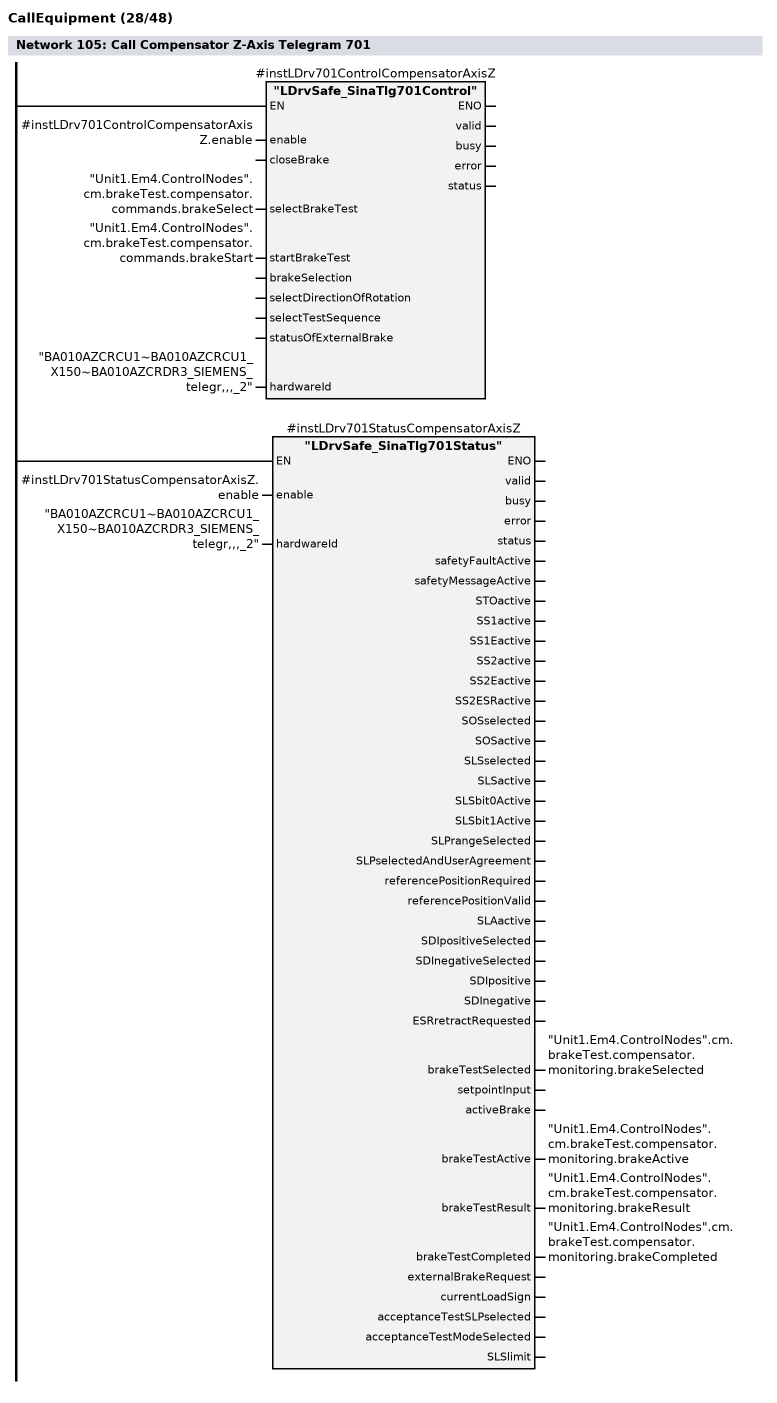
   RUNG wire#powerrail
      #instLDrv701ControlCompensatorAxisZ(enable := #instLDrv701ControlCompensatorAxisZ.enable, closeBrake :=, selectBrakeTest := "Unit1.Em4.ControlNodes".cm.brakeTest.compensator.commands.brakeSelect, startBrakeTest := "Unit1.Em4.ControlNodes".cm.brakeTest.compensator.commands.brakeStart, brakeSelection :=, selectDirectionOfRotation :=, selectTestSequence :=, statusOfExternalBrake :=, hardwareId := "BA010AZCRCU1~BA010AZCRCU1_X150~BA010AZCRDR3_SIEMENS_telegr,,,_2", valid =>, busy =>, error =>, status =>)
   END_RUNG
   RUNG wire#powerrail
      #instLDrv701StatusCompensatorAxisZ(enable := #instLDrv701StatusCompensatorAxisZ.enable, hardwareId := "BA010AZCRCU1~BA010AZCRCU1_X150~BA010AZCRDR3_SIEMENS_telegr,,,_2", valid =>, busy =>, error =>, status =>, safetyFaultActive =>, safetyMessageActive =>, STOactive =>, SS1active =>, SS1Eactive =>, SS2active =>, SS2Eactive =>, SS2ESRactive =>, SOSselected =>, SOSactive =>, SLSselected =>, SLSactive =>, SLSbit0Active =>, SLSbit1Active =>, SLPrangeSelected =>, SLPselectedAndUserAgreement =>, referencePositionRequired =>, referencePositionValid =>, SLAactive =>, SDIpositiveSelected =>, SDInegativeSelected =>, SDIpositive =>, SDInegative =>, ESRretractRequested =>, brakeTestSelected => "Unit1.Em4.ControlNodes".cm.brakeTest.compensator.monitoring.brakeSelected, setpointInput =>, activeBrake =>, brakeTestActive => "Unit1.Em4.ControlNodes".cm.brakeTest.compensator.monitoring.brakeActive, brakeTestResult => "Unit1.Em4.ControlNodes".cm.brakeTest.compensator.monitoring.brakeResult, brakeTestCompleted => "Unit1.Em4.ControlNodes".cm.brakeTest.compensator.monitoring.brakeCompleted, externalBrakeRequest =>, currentLoadSign =>, acceptanceTestSLPselected =>, acceptanceTestModeSelected =>, SLSlimit =>)
   END_RUNG
   // the same network as SCL:
   #instLDrv701ControlCompensatorAxisZ(enable := #instLDrv701ControlCompensatorAxisZ.enable,   // "LDrvSafe_SinaTlg701Control"
                           selectBrakeTest := "Unit1.Em4.ControlNodes".cm.brakeTest.compensator.commands.brakeSelect,
                           startBrakeTest := "Unit1.Em4.ControlNodes".cm.brakeTest.compensator.commands.brakeStart,
                           hardwareId := "BA010AZCRCU1~BA010AZCRCU1_X150~BA010AZCRDR3_SIEMENS_telegr,,,_2");
   #instLDrv701StatusCompensatorAxisZ(enable := #instLDrv701StatusCompensatorAxisZ.enable,   // "LDrvSafe_SinaTlg701Status"
                           hardwareId := "BA010AZCRCU1~BA010AZCRCU1_X150~BA010AZCRDR3_SIEMENS_telegr,,,_2",
                           brakeTestSelected => "Unit1.Em4.ControlNodes".cm.brakeTest.compensator.monitoring.brakeSelected,
                           brakeTestActive => "Unit1.Em4.ControlNodes".cm.brakeTest.compensator.monitoring.brakeActive,
                           brakeTestResult => "Unit1.Em4.ControlNodes".cm.brakeTest.compensator.monitoring.brakeResult,
                           brakeTestCompleted => "Unit1.Em4.ControlNodes".cm.brakeTest.compensator.monitoring.brakeCompleted);
END_REGION

REGION Network 107: FeedingRoll B-Axis Brake Test Error
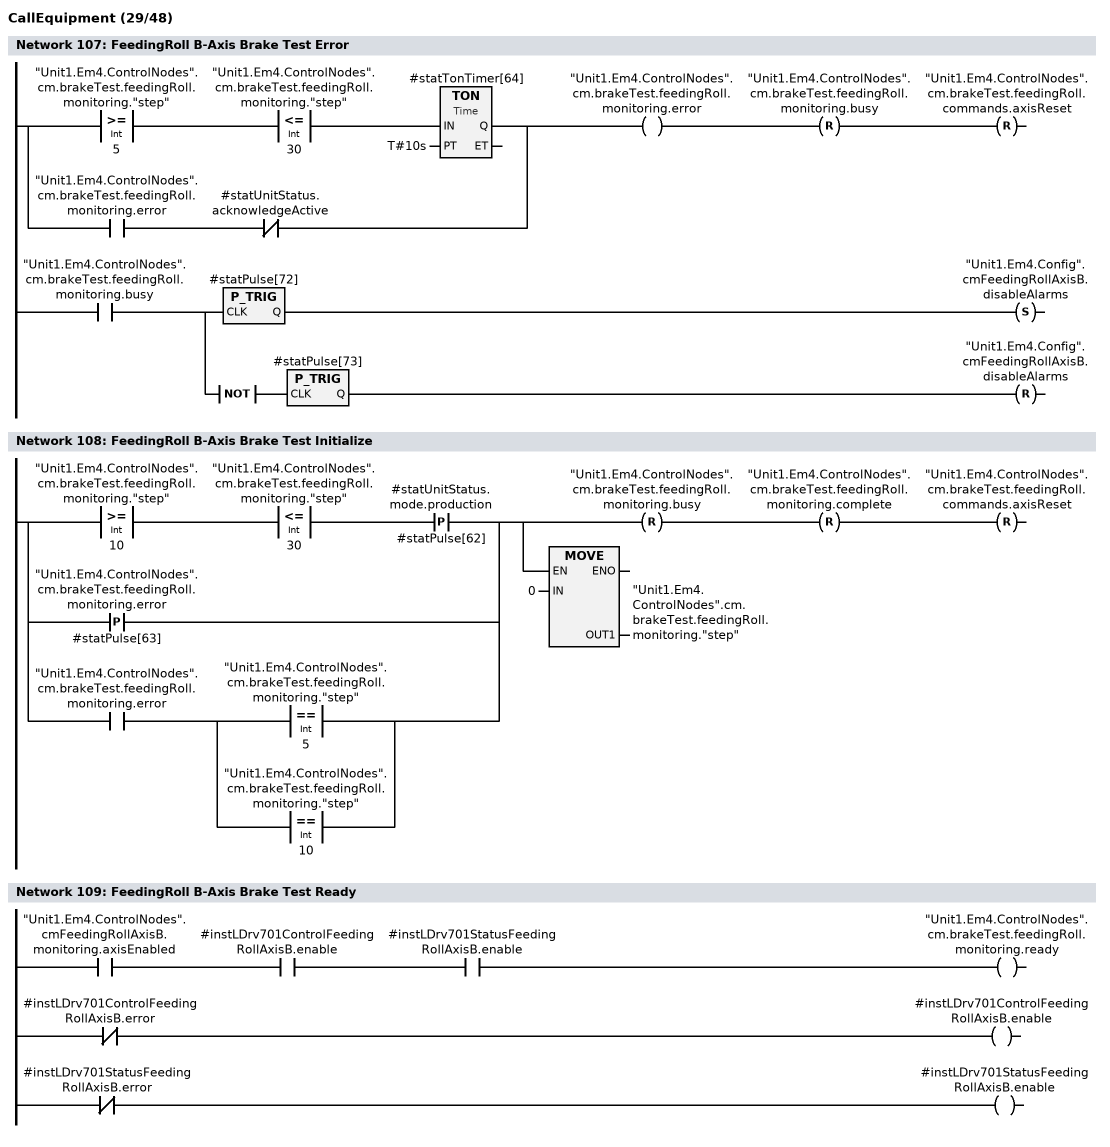
   RUNG wire#powerrail
      { S7_Templates := "SrcType := Int" } GE_Contact(in1 := "Unit1.Em4.ControlNodes".cm.brakeTest.feedingRoll.monitoring."step", in2 := 5)
      { S7_Templates := "SrcType := Int" } LE_Contact(in1 := "Unit1.Em4.ControlNodes".cm.brakeTest.feedingRoll.monitoring."step", in2 := 30)
      { S7_Templates := "time_type := Time" } #statTonTimer[64].TON(pt := T#10s, et =>)
      wire#w1
      Coil( "Unit1.Em4.ControlNodes".cm.brakeTest.feedingRoll.monitoring.error )
      R_Coil( "Unit1.Em4.ControlNodes".cm.brakeTest.feedingRoll.monitoring.busy )
      R_Coil( "Unit1.Em4.ControlNodes".cm.brakeTest.feedingRoll.commands.axisReset )
   END_RUNG
   RUNG wire#powerrail
      Contact( "Unit1.Em4.ControlNodes".cm.brakeTest.feedingRoll.monitoring.error )
      I_Contact( #statUnitStatus.acknowledgeActive )
   END_RUNG wire#w1
   RUNG wire#powerrail
      Contact( "Unit1.Em4.ControlNodes".cm.brakeTest.feedingRoll.monitoring.busy )
      wire#w2
      P_Trig( #statPulse[72] )
      S_Coil( "Unit1.Em4.Config".cmFeedingRollAxisB.disableAlarms )
   END_RUNG
   RUNG wire#w2
      Not()
      P_Trig( #statPulse[73] )
      R_Coil( "Unit1.Em4.Config".cmFeedingRollAxisB.disableAlarms )
   END_RUNG
   // the same network as SCL:
   #statTonTimer[64].TON(IN := ("Unit1.Em4.ControlNodes".cm.brakeTest.feedingRoll.monitoring."step" >= 5) AND ("Unit1.Em4.ControlNodes".cm.brakeTest.feedingRoll.monitoring."step" <= 30),
                         PT := T#10s);
   "Unit1.Em4.ControlNodes".cm.brakeTest.feedingRoll.monitoring.error := #statTonTimer[64].Q OR ("Unit1.Em4.ControlNodes".cm.brakeTest.feedingRoll.monitoring.error AND NOT #statUnitStatus.acknowledgeActive);
   IF "Unit1.Em4.ControlNodes".cm.brakeTest.feedingRoll.monitoring.error THEN
       "Unit1.Em4.ControlNodes".cm.brakeTest.feedingRoll.monitoring.busy := FALSE;
       "Unit1.Em4.ControlNodes".cm.brakeTest.feedingRoll.commands.axisReset := FALSE;
   END_IF;
   #_w1 := "Unit1.Em4.ControlNodes".cm.brakeTest.feedingRoll.monitoring.busy AND NOT #statPulse[72];   // rising edge
   #statPulse[72] := "Unit1.Em4.ControlNodes".cm.brakeTest.feedingRoll.monitoring.busy;
   IF #_w1 THEN "Unit1.Em4.Config".cmFeedingRollAxisB.disableAlarms := TRUE; END_IF;
   #_w2 := NOT "Unit1.Em4.ControlNodes".cm.brakeTest.feedingRoll.monitoring.busy AND NOT #statPulse[73];   // rising edge
   #statPulse[73] := NOT "Unit1.Em4.ControlNodes".cm.brakeTest.feedingRoll.monitoring.busy;
   IF #_w2 THEN "Unit1.Em4.Config".cmFeedingRollAxisB.disableAlarms := FALSE; END_IF;
END_REGION

REGION Network 108: FeedingRoll B-Axis Brake Test Initialize
   RUNG wire#powerrail
      { S7_Templates := "SrcType := Int" } GE_Contact(in1 := "Unit1.Em4.ControlNodes".cm.brakeTest.feedingRoll.monitoring."step", in2 := 10)
      { S7_Templates := "SrcType := Int" } LE_Contact(in1 := "Unit1.Em4.ControlNodes".cm.brakeTest.feedingRoll.monitoring."step", in2 := 30)
      P_Contact(operand := #statUnitStatus.mode.production, bit := #statPulse[62])
      wire#w1
      R_Coil( "Unit1.Em4.ControlNodes".cm.brakeTest.feedingRoll.monitoring.busy )
      R_Coil( "Unit1.Em4.ControlNodes".cm.brakeTest.feedingRoll.monitoring.complete )
      R_Coil( "Unit1.Em4.ControlNodes".cm.brakeTest.feedingRoll.commands.axisReset )
   END_RUNG
   RUNG wire#powerrail
      P_Contact(operand := "Unit1.Em4.ControlNodes".cm.brakeTest.feedingRoll.monitoring.error, bit := #statPulse[63])
   END_RUNG wire#w1
   RUNG wire#powerrail
      Contact( "Unit1.Em4.ControlNodes".cm.brakeTest.feedingRoll.monitoring.error )
      wire#w2
      { S7_Templates := "SrcType := Int" } EQ_Contact(in1 := "Unit1.Em4.ControlNodes".cm.brakeTest.feedingRoll.monitoring."step", in2 := 5)
   END_RUNG wire#w1
   RUNG wire#w2
      { S7_Templates := "SrcType := Int" } EQ_Contact(in1 := "Unit1.Em4.ControlNodes".cm.brakeTest.feedingRoll.monitoring."step", in2 := 10)
   END_RUNG wire#w1
   RUNG wire#w1
      Move(in := 0, out1 => "Unit1.Em4.ControlNodes".cm.brakeTest.feedingRoll.monitoring."step")
   END_RUNG
   // the same network as SCL:
   #_w1 := ("Unit1.Em4.ControlNodes".cm.brakeTest.feedingRoll.monitoring."step" >= 10) AND ("Unit1.Em4.ControlNodes".cm.brakeTest.feedingRoll.monitoring."step" <= 30) AND #statUnitStatus.mode.production AND NOT #statPulse[62];   // rising edge of #statUnitStatus.mode.production
   #statPulse[62] := #statUnitStatus.mode.production;
   #_w2 := "Unit1.Em4.ControlNodes".cm.brakeTest.feedingRoll.monitoring.error AND NOT #statPulse[63];   // rising edge of "Unit1.Em4.ControlNodes".cm.brakeTest.feedingRoll.monitoring.error
   #statPulse[63] := "Unit1.Em4.ControlNodes".cm.brakeTest.feedingRoll.monitoring.error;
   IF #_w1 OR #_w2 OR ("Unit1.Em4.ControlNodes".cm.brakeTest.feedingRoll.monitoring.error AND (("Unit1.Em4.ControlNodes".cm.brakeTest.feedingRoll.monitoring."step" = 5) OR ("Unit1.Em4.ControlNodes".cm.brakeTest.feedingRoll.monitoring."step" = 10))) THEN
       "Unit1.Em4.ControlNodes".cm.brakeTest.feedingRoll.monitoring.busy := FALSE;
       "Unit1.Em4.ControlNodes".cm.brakeTest.feedingRoll.monitoring.complete := FALSE;
       "Unit1.Em4.ControlNodes".cm.brakeTest.feedingRoll.commands.axisReset := FALSE;
       "Unit1.Em4.ControlNodes".cm.brakeTest.feedingRoll.monitoring."step" := 0;
   END_IF;
END_REGION

REGION Network 109: FeedingRoll B-Axis Brake Test Ready
   RUNG wire#powerrail
      Contact( "Unit1.Em4.ControlNodes".cmFeedingRollAxisB.monitoring.axisEnabled )
      Contact( #instLDrv701ControlFeedingRollAxisB.enable )
      Contact( #instLDrv701StatusFeedingRollAxisB.enable )
      Coil( "Unit1.Em4.ControlNodes".cm.brakeTest.feedingRoll.monitoring.ready )
   END_RUNG
   RUNG wire#powerrail
      I_Contact( #instLDrv701ControlFeedingRollAxisB.error )
      Coil( #instLDrv701ControlFeedingRollAxisB.enable )
   END_RUNG
   RUNG wire#powerrail
      I_Contact( #instLDrv701StatusFeedingRollAxisB.error )
      Coil( #instLDrv701StatusFeedingRollAxisB.enable )
   END_RUNG
   // the same network as SCL:
   "Unit1.Em4.ControlNodes".cm.brakeTest.feedingRoll.monitoring.ready := "Unit1.Em4.ControlNodes".cmFeedingRollAxisB.monitoring.axisEnabled AND #instLDrv701ControlFeedingRollAxisB.enable AND #instLDrv701StatusFeedingRollAxisB.enable;
   #instLDrv701ControlFeedingRollAxisB.enable := NOT #instLDrv701ControlFeedingRollAxisB.error;
   #instLDrv701StatusFeedingRollAxisB.enable := NOT #instLDrv701StatusFeedingRollAxisB.error;
END_REGION

REGION Network 110: FeedingRoll B-Axis Reset
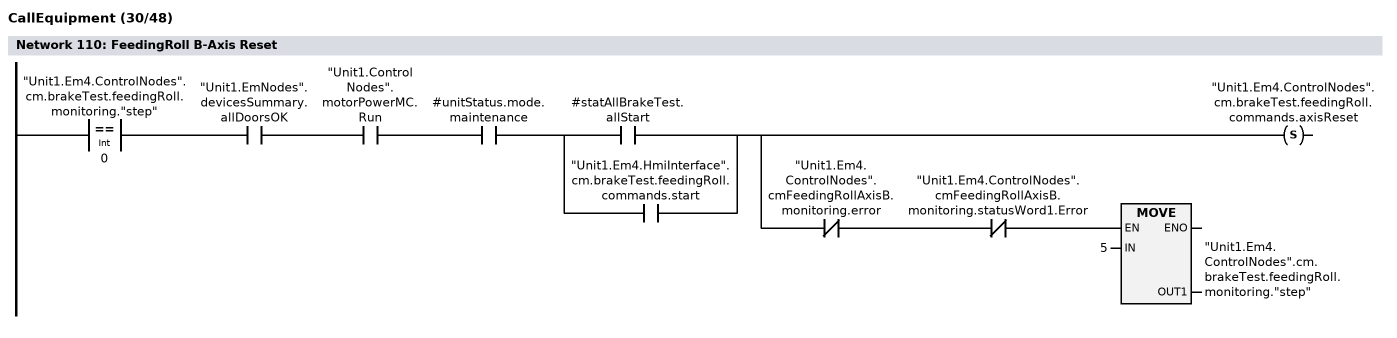
   RUNG wire#powerrail
      { S7_Templates := "SrcType := Int" } EQ_Contact(in1 := "Unit1.Em4.ControlNodes".cm.brakeTest.feedingRoll.monitoring."step", in2 := 0)
      Contact( "Unit1.EmNodes".devicesSummary.allDoorsOK )
      Contact( "Unit1.ControlNodes".motorPowerMC.Run )
      Contact( #unitStatus.mode.maintenance )
      wire#w1
      Contact( #statAllBrakeTest.allStart )
      wire#w2
      S_Coil( "Unit1.Em4.ControlNodes".cm.brakeTest.feedingRoll.commands.axisReset )
   END_RUNG
   RUNG wire#w1
      Contact( "Unit1.Em4.HmiInterface".cm.brakeTest.feedingRoll.commands.start )
   END_RUNG wire#w2
   RUNG wire#w2
      I_Contact( "Unit1.Em4.ControlNodes".cmFeedingRollAxisB.monitoring.error )
      I_Contact( "Unit1.Em4.ControlNodes".cmFeedingRollAxisB.monitoring.statusWord1.Error )
      Move(in := 5, out1 => "Unit1.Em4.ControlNodes".cm.brakeTest.feedingRoll.monitoring."step")
   END_RUNG
   // the same network as SCL:
   #_w1 := ("Unit1.Em4.ControlNodes".cm.brakeTest.feedingRoll.monitoring."step" = 0) AND "Unit1.EmNodes".devicesSummary.allDoorsOK AND "Unit1.ControlNodes".motorPowerMC.Run AND #unitStatus.mode.maintenance AND (#statAllBrakeTest.allStart OR "Unit1.Em4.HmiInterface".cm.brakeTest.feedingRoll.commands.start);
   IF #_w1 THEN "Unit1.Em4.ControlNodes".cm.brakeTest.feedingRoll.commands.axisReset := TRUE; END_IF;
   IF #_w1 AND NOT "Unit1.Em4.ControlNodes".cmFeedingRollAxisB.monitoring.error AND NOT "Unit1.Em4.ControlNodes".cmFeedingRollAxisB.monitoring.statusWord1.Error THEN
       "Unit1.Em4.ControlNodes".cm.brakeTest.feedingRoll.monitoring."step" := 5;
   END_IF;
END_REGION

REGION Network 111: FeedingRoll B-Axis Brake Test Commands
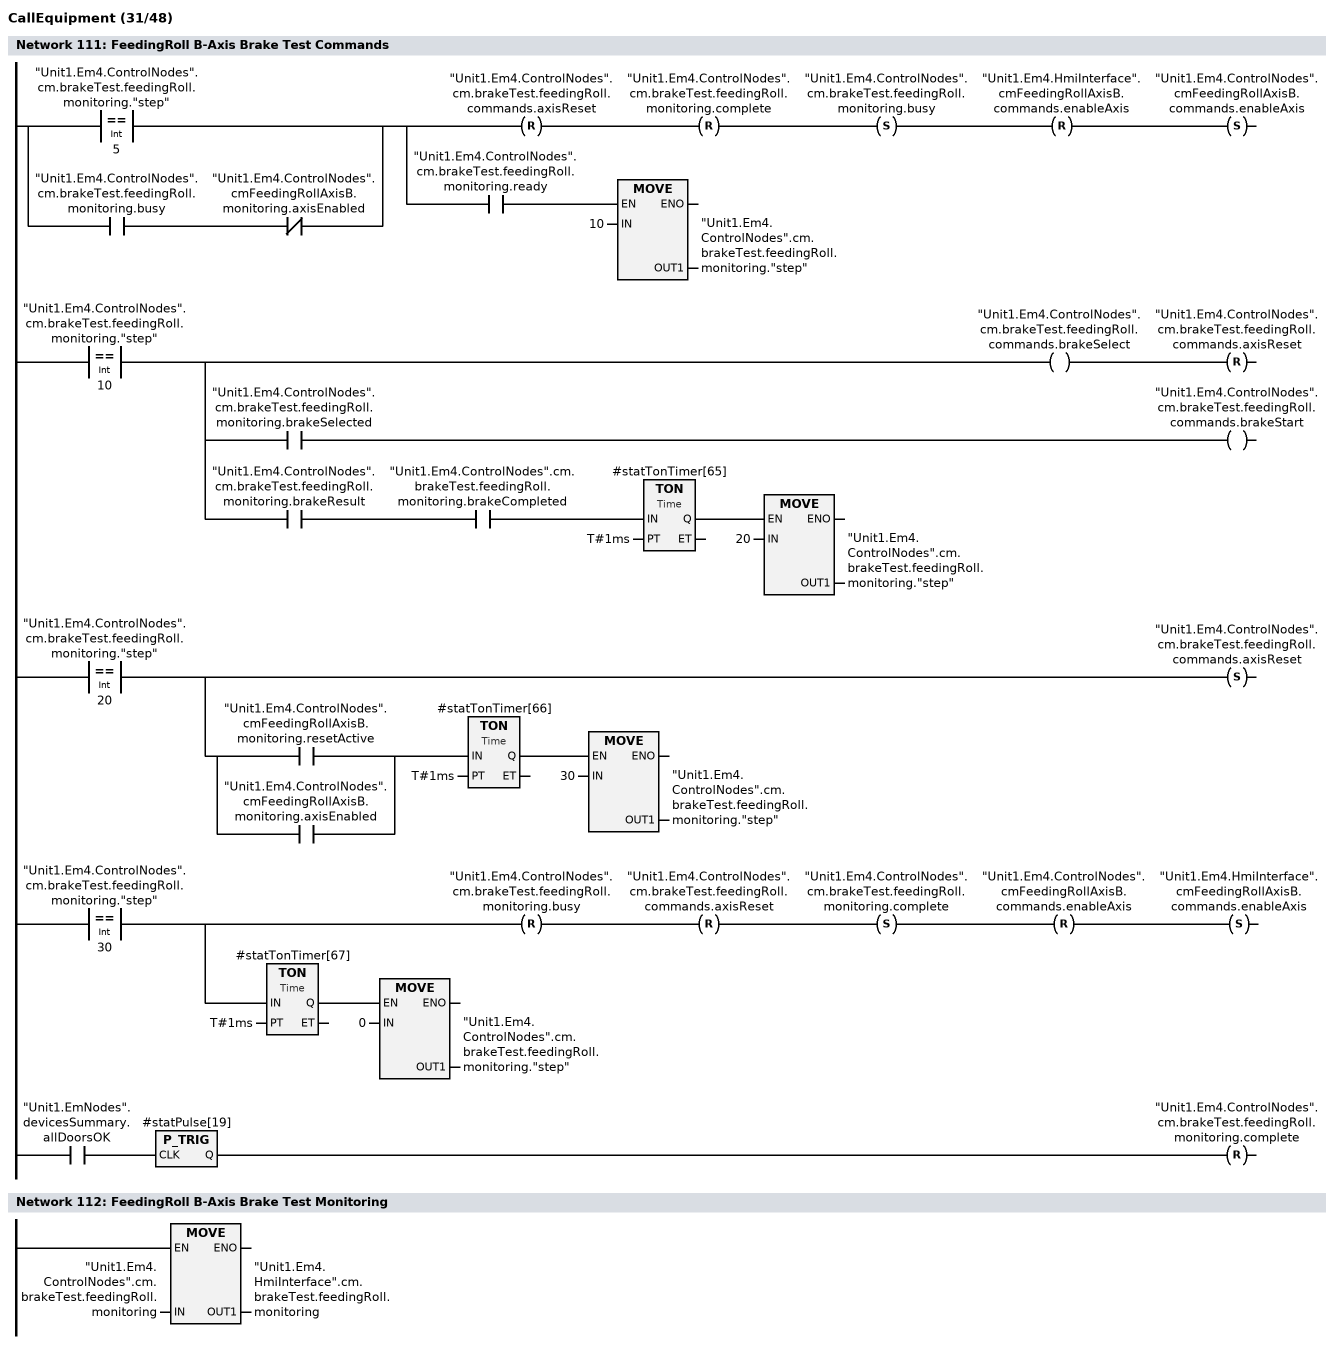
   RUNG wire#powerrail
      { S7_Templates := "SrcType := Int" } EQ_Contact(in1 := "Unit1.Em4.ControlNodes".cm.brakeTest.feedingRoll.monitoring."step", in2 := 5)
      wire#w1
      R_Coil( "Unit1.Em4.ControlNodes".cm.brakeTest.feedingRoll.commands.axisReset )
      R_Coil( "Unit1.Em4.ControlNodes".cm.brakeTest.feedingRoll.monitoring.complete )
      S_Coil( "Unit1.Em4.ControlNodes".cm.brakeTest.feedingRoll.monitoring.busy )
      R_Coil( "Unit1.Em4.HmiInterface".cmFeedingRollAxisB.commands.enableAxis )
      S_Coil( "Unit1.Em4.ControlNodes".cmFeedingRollAxisB.commands.enableAxis )
   END_RUNG
   RUNG wire#powerrail
      Contact( "Unit1.Em4.ControlNodes".cm.brakeTest.feedingRoll.monitoring.busy )
      I_Contact( "Unit1.Em4.ControlNodes".cmFeedingRollAxisB.monitoring.axisEnabled )
   END_RUNG wire#w1
   RUNG wire#w1
      Contact( "Unit1.Em4.ControlNodes".cm.brakeTest.feedingRoll.monitoring.ready )
      Move(in := 10, out1 => "Unit1.Em4.ControlNodes".cm.brakeTest.feedingRoll.monitoring."step")
   END_RUNG
   RUNG wire#powerrail
      { S7_Templates := "SrcType := Int" } EQ_Contact(in1 := "Unit1.Em4.ControlNodes".cm.brakeTest.feedingRoll.monitoring."step", in2 := 10)
      wire#w2
      Coil( "Unit1.Em4.ControlNodes".cm.brakeTest.feedingRoll.commands.brakeSelect )
      R_Coil( "Unit1.Em4.ControlNodes".cm.brakeTest.feedingRoll.commands.axisReset )
   END_RUNG
   RUNG wire#w2
      Contact( "Unit1.Em4.ControlNodes".cm.brakeTest.feedingRoll.monitoring.brakeSelected )
      Coil( "Unit1.Em4.ControlNodes".cm.brakeTest.feedingRoll.commands.brakeStart )
   END_RUNG
   RUNG wire#w2
      Contact( "Unit1.Em4.ControlNodes".cm.brakeTest.feedingRoll.monitoring.brakeResult )
      Contact( "Unit1.Em4.ControlNodes".cm.brakeTest.feedingRoll.monitoring.brakeCompleted )
      { S7_Templates := "time_type := Time" } #statTonTimer[65].TON(pt := T#1ms, et =>)
      Move(in := 20, out1 => "Unit1.Em4.ControlNodes".cm.brakeTest.feedingRoll.monitoring."step")
   END_RUNG
   RUNG wire#powerrail
      { S7_Templates := "SrcType := Int" } EQ_Contact(in1 := "Unit1.Em4.ControlNodes".cm.brakeTest.feedingRoll.monitoring."step", in2 := 20)
      wire#w3
      S_Coil( "Unit1.Em4.ControlNodes".cm.brakeTest.feedingRoll.commands.axisReset )
   END_RUNG
   RUNG wire#w3
      Contact( "Unit1.Em4.ControlNodes".cmFeedingRollAxisB.monitoring.resetActive )
      wire#w4
      { S7_Templates := "time_type := Time" } #statTonTimer[66].TON(pt := T#1ms, et =>)
      Move(in := 30, out1 => "Unit1.Em4.ControlNodes".cm.brakeTest.feedingRoll.monitoring."step")
   END_RUNG
   RUNG wire#w3
      Contact( "Unit1.Em4.ControlNodes".cmFeedingRollAxisB.monitoring.axisEnabled )
   END_RUNG wire#w4
   RUNG wire#powerrail
      { S7_Templates := "SrcType := Int" } EQ_Contact(in1 := "Unit1.Em4.ControlNodes".cm.brakeTest.feedingRoll.monitoring."step", in2 := 30)
      wire#w5
      R_Coil( "Unit1.Em4.ControlNodes".cm.brakeTest.feedingRoll.monitoring.busy )
      R_Coil( "Unit1.Em4.ControlNodes".cm.brakeTest.feedingRoll.commands.axisReset )
      S_Coil( "Unit1.Em4.ControlNodes".cm.brakeTest.feedingRoll.monitoring.complete )
      R_Coil( "Unit1.Em4.ControlNodes".cmFeedingRollAxisB.commands.enableAxis )
      S_Coil( "Unit1.Em4.HmiInterface".cmFeedingRollAxisB.commands.enableAxis )
   END_RUNG
   RUNG wire#w5
      { S7_Templates := "time_type := Time" } #statTonTimer[67].TON(pt := T#1ms, et =>)
      Move(in := 0, out1 => "Unit1.Em4.ControlNodes".cm.brakeTest.feedingRoll.monitoring."step")
   END_RUNG
   RUNG wire#powerrail
      Contact( "Unit1.EmNodes".devicesSummary.allDoorsOK )
      P_Trig( #statPulse[19] )
      R_Coil( "Unit1.Em4.ControlNodes".cm.brakeTest.feedingRoll.monitoring.complete )
   END_RUNG
   // the same network as SCL:
   #_w1 := ("Unit1.Em4.ControlNodes".cm.brakeTest.feedingRoll.monitoring."step" = 5) OR ("Unit1.Em4.ControlNodes".cm.brakeTest.feedingRoll.monitoring.busy AND NOT "Unit1.Em4.ControlNodes".cmFeedingRollAxisB.monitoring.axisEnabled);
   IF #_w1 THEN
       "Unit1.Em4.ControlNodes".cm.brakeTest.feedingRoll.commands.axisReset := FALSE;
       "Unit1.Em4.ControlNodes".cm.brakeTest.feedingRoll.monitoring.complete := FALSE;
       "Unit1.Em4.ControlNodes".cm.brakeTest.feedingRoll.monitoring.busy := TRUE;
       "Unit1.Em4.HmiInterface".cmFeedingRollAxisB.commands.enableAxis := FALSE;
       "Unit1.Em4.ControlNodes".cmFeedingRollAxisB.commands.enableAxis := TRUE;
   END_IF;
   IF #_w1 AND "Unit1.Em4.ControlNodes".cm.brakeTest.feedingRoll.monitoring.ready THEN
       "Unit1.Em4.ControlNodes".cm.brakeTest.feedingRoll.monitoring."step" := 10;
   END_IF;
   "Unit1.Em4.ControlNodes".cm.brakeTest.feedingRoll.commands.brakeSelect := "Unit1.Em4.ControlNodes".cm.brakeTest.feedingRoll.monitoring."step" = 10;
   IF "Unit1.Em4.ControlNodes".cm.brakeTest.feedingRoll.commands.brakeSelect THEN
       "Unit1.Em4.ControlNodes".cm.brakeTest.feedingRoll.commands.axisReset := FALSE;
   END_IF;
   "Unit1.Em4.ControlNodes".cm.brakeTest.feedingRoll.commands.brakeStart := "Unit1.Em4.ControlNodes".cm.brakeTest.feedingRoll.commands.brakeSelect AND "Unit1.Em4.ControlNodes".cm.brakeTest.feedingRoll.monitoring.brakeSelected;
   #statTonTimer[65].TON(IN := "Unit1.Em4.ControlNodes".cm.brakeTest.feedingRoll.commands.brakeSelect AND "Unit1.Em4.ControlNodes".cm.brakeTest.feedingRoll.monitoring.brakeResult AND "Unit1.Em4.ControlNodes".cm.brakeTest.feedingRoll.monitoring.brakeCompleted,
                         PT := T#1ms);
   IF #statTonTimer[65].Q THEN
       "Unit1.Em4.ControlNodes".cm.brakeTest.feedingRoll.monitoring."step" := 20;
   END_IF;
   #_w2 := "Unit1.Em4.ControlNodes".cm.brakeTest.feedingRoll.monitoring."step" = 20;
   IF #_w2 THEN "Unit1.Em4.ControlNodes".cm.brakeTest.feedingRoll.commands.axisReset := TRUE; END_IF;
   #statTonTimer[66].TON(IN := #_w2 AND ("Unit1.Em4.ControlNodes".cmFeedingRollAxisB.monitoring.resetActive OR "Unit1.Em4.ControlNodes".cmFeedingRollAxisB.monitoring.axisEnabled),
                         PT := T#1ms);
   IF #statTonTimer[66].Q THEN
       "Unit1.Em4.ControlNodes".cm.brakeTest.feedingRoll.monitoring."step" := 30;
   END_IF;
   #_w3 := "Unit1.Em4.ControlNodes".cm.brakeTest.feedingRoll.monitoring."step" = 30;
   IF #_w3 THEN
       "Unit1.Em4.ControlNodes".cm.brakeTest.feedingRoll.monitoring.busy := FALSE;
       "Unit1.Em4.ControlNodes".cm.brakeTest.feedingRoll.commands.axisReset := FALSE;
       "Unit1.Em4.ControlNodes".cm.brakeTest.feedingRoll.monitoring.complete := TRUE;
       "Unit1.Em4.ControlNodes".cmFeedingRollAxisB.commands.enableAxis := FALSE;
       "Unit1.Em4.HmiInterface".cmFeedingRollAxisB.commands.enableAxis := TRUE;
   END_IF;
   #statTonTimer[67].TON(IN := #_w3, PT := T#1ms);
   IF #statTonTimer[67].Q THEN
       "Unit1.Em4.ControlNodes".cm.brakeTest.feedingRoll.monitoring."step" := 0;
   END_IF;
   #_w4 := "Unit1.EmNodes".devicesSummary.allDoorsOK AND NOT #statPulse[19];   // rising edge
   #statPulse[19] := "Unit1.EmNodes".devicesSummary.allDoorsOK;
   IF #_w4 THEN "Unit1.Em4.ControlNodes".cm.brakeTest.feedingRoll.monitoring.complete := FALSE; END_IF;
END_REGION

REGION Network 112: FeedingRoll B-Axis Brake Test Monitoring
   RUNG wire#powerrail
      Move(in := "Unit1.Em4.ControlNodes".cm.brakeTest.feedingRoll.monitoring, out1 => "Unit1.Em4.HmiInterface".cm.brakeTest.feedingRoll.monitoring)
   END_RUNG
   // the same network as SCL:
   "Unit1.Em4.HmiInterface".cm.brakeTest.feedingRoll.monitoring := "Unit1.Em4.ControlNodes".cm.brakeTest.feedingRoll.monitoring;
END_REGION

REGION Network 113: Call FeedingRoll B-Axis Telegram 701
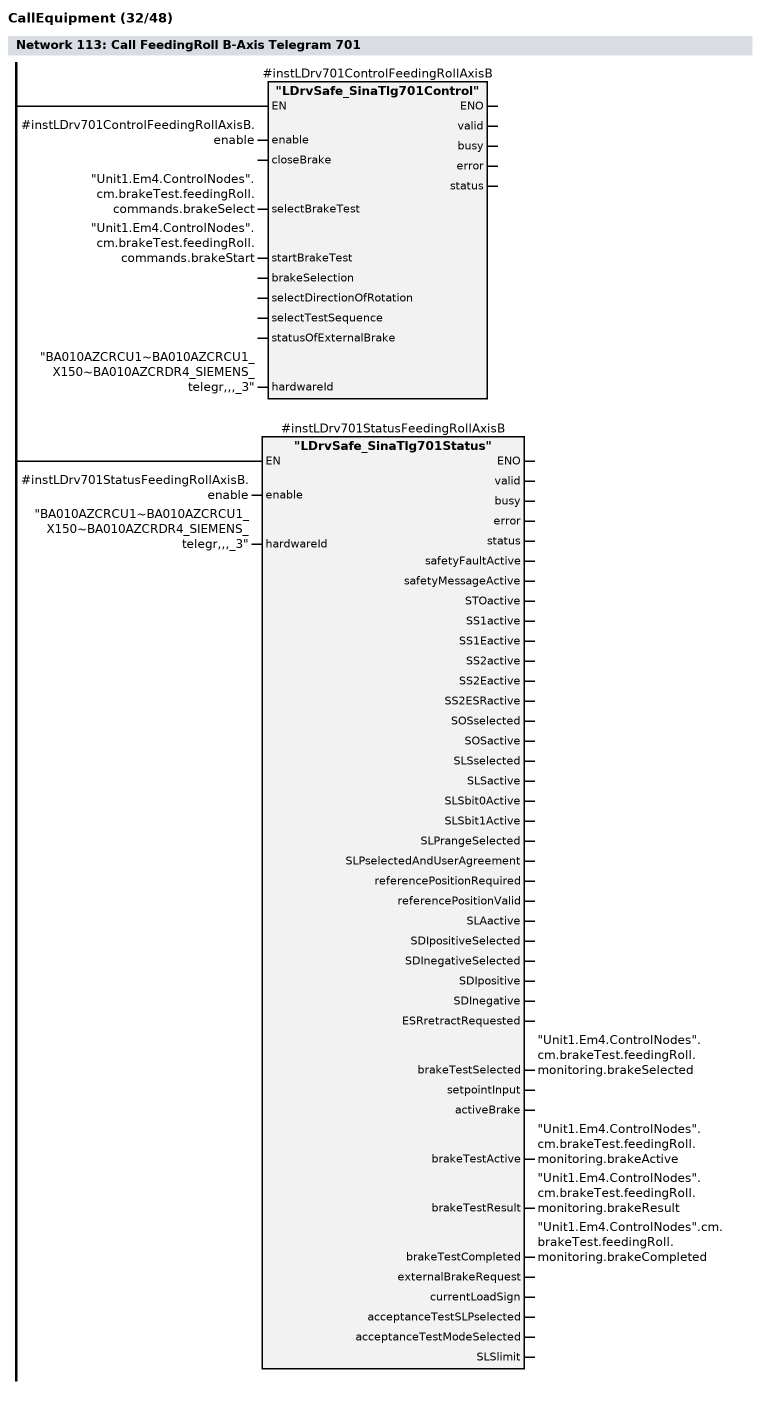
   RUNG wire#powerrail
      #instLDrv701ControlFeedingRollAxisB(enable := #instLDrv701ControlFeedingRollAxisB.enable, closeBrake :=, selectBrakeTest := "Unit1.Em4.ControlNodes".cm.brakeTest.feedingRoll.commands.brakeSelect, startBrakeTest := "Unit1.Em4.ControlNodes".cm.brakeTest.feedingRoll.commands.brakeStart, brakeSelection :=, selectDirectionOfRotation :=, selectTestSequence :=, statusOfExternalBrake :=, hardwareId := "BA010AZCRCU1~BA010AZCRCU1_X150~BA010AZCRDR4_SIEMENS_telegr,,,_3", valid =>, busy =>, error =>, status =>)
   END_RUNG
   RUNG wire#powerrail
      #instLDrv701StatusFeedingRollAxisB(enable := #instLDrv701StatusFeedingRollAxisB.enable, hardwareId := "BA010AZCRCU1~BA010AZCRCU1_X150~BA010AZCRDR4_SIEMENS_telegr,,,_3", valid =>, busy =>, error =>, status =>, safetyFaultActive =>, safetyMessageActive =>, STOactive =>, SS1active =>, SS1Eactive =>, SS2active =>, SS2Eactive =>, SS2ESRactive =>, SOSselected =>, SOSactive =>, SLSselected =>, SLSactive =>, SLSbit0Active =>, SLSbit1Active =>, SLPrangeSelected =>, SLPselectedAndUserAgreement =>, referencePositionRequired =>, referencePositionValid =>, SLAactive =>, SDIpositiveSelected =>, SDInegativeSelected =>, SDIpositive =>, SDInegative =>, ESRretractRequested =>, brakeTestSelected => "Unit1.Em4.ControlNodes".cm.brakeTest.feedingRoll.monitoring.brakeSelected, setpointInput =>, activeBrake =>, brakeTestActive => "Unit1.Em4.ControlNodes".cm.brakeTest.feedingRoll.monitoring.brakeActive, brakeTestResult => "Unit1.Em4.ControlNodes".cm.brakeTest.feedingRoll.monitoring.brakeResult, brakeTestCompleted => "Unit1.Em4.ControlNodes".cm.brakeTest.feedingRoll.monitoring.brakeCompleted, externalBrakeRequest =>, currentLoadSign =>, acceptanceTestSLPselected =>, acceptanceTestModeSelected =>, SLSlimit =>)
   END_RUNG
   // the same network as SCL:
   #instLDrv701ControlFeedingRollAxisB(enable := #instLDrv701ControlFeedingRollAxisB.enable,   // "LDrvSafe_SinaTlg701Control"
                           selectBrakeTest := "Unit1.Em4.ControlNodes".cm.brakeTest.feedingRoll.commands.brakeSelect,
                           startBrakeTest := "Unit1.Em4.ControlNodes".cm.brakeTest.feedingRoll.commands.brakeStart,
                           hardwareId := "BA010AZCRCU1~BA010AZCRCU1_X150~BA010AZCRDR4_SIEMENS_telegr,,,_3");
   #instLDrv701StatusFeedingRollAxisB(enable := #instLDrv701StatusFeedingRollAxisB.enable,   // "LDrvSafe_SinaTlg701Status"
                           hardwareId := "BA010AZCRCU1~BA010AZCRCU1_X150~BA010AZCRDR4_SIEMENS_telegr,,,_3",
                           brakeTestSelected => "Unit1.Em4.ControlNodes".cm.brakeTest.feedingRoll.monitoring.brakeSelected,
                           brakeTestActive => "Unit1.Em4.ControlNodes".cm.brakeTest.feedingRoll.monitoring.brakeActive,
                           brakeTestResult => "Unit1.Em4.ControlNodes".cm.brakeTest.feedingRoll.monitoring.brakeResult,
                           brakeTestCompleted => "Unit1.Em4.ControlNodes".cm.brakeTest.feedingRoll.monitoring.brakeCompleted);
END_REGION

REGION Network 115: Cutter Z-Axis Brake Test Error
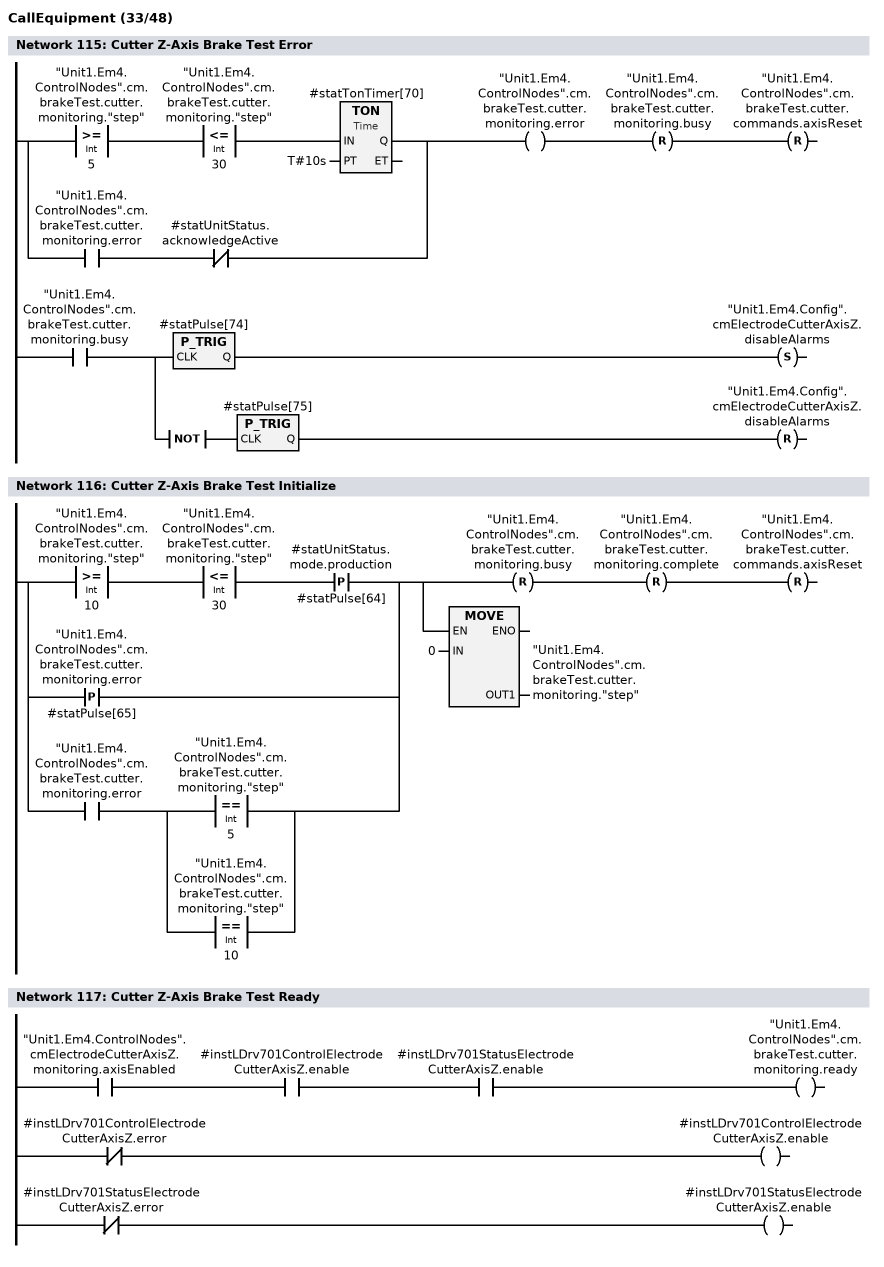
   RUNG wire#powerrail
      { S7_Templates := "SrcType := Int" } GE_Contact(in1 := "Unit1.Em4.ControlNodes".cm.brakeTest.cutter.monitoring."step", in2 := 5)
      { S7_Templates := "SrcType := Int" } LE_Contact(in1 := "Unit1.Em4.ControlNodes".cm.brakeTest.cutter.monitoring."step", in2 := 30)
      { S7_Templates := "time_type := Time" } #statTonTimer[70].TON(pt := T#10s, et =>)
      wire#w1
      Coil( "Unit1.Em4.ControlNodes".cm.brakeTest.cutter.monitoring.error )
      R_Coil( "Unit1.Em4.ControlNodes".cm.brakeTest.cutter.monitoring.busy )
      R_Coil( "Unit1.Em4.ControlNodes".cm.brakeTest.cutter.commands.axisReset )
   END_RUNG
   RUNG wire#powerrail
      Contact( "Unit1.Em4.ControlNodes".cm.brakeTest.cutter.monitoring.error )
      I_Contact( #statUnitStatus.acknowledgeActive )
   END_RUNG wire#w1
   RUNG wire#powerrail
      Contact( "Unit1.Em4.ControlNodes".cm.brakeTest.cutter.monitoring.busy )
      wire#w2
      P_Trig( #statPulse[74] )
      S_Coil( "Unit1.Em4.Config".cmElectrodeCutterAxisZ.disableAlarms )
   END_RUNG
   RUNG wire#w2
      Not()
      P_Trig( #statPulse[75] )
      R_Coil( "Unit1.Em4.Config".cmElectrodeCutterAxisZ.disableAlarms )
   END_RUNG
   // the same network as SCL:
   #statTonTimer[70].TON(IN := ("Unit1.Em4.ControlNodes".cm.brakeTest.cutter.monitoring."step" >= 5) AND ("Unit1.Em4.ControlNodes".cm.brakeTest.cutter.monitoring."step" <= 30),
                         PT := T#10s);
   "Unit1.Em4.ControlNodes".cm.brakeTest.cutter.monitoring.error := #statTonTimer[70].Q OR ("Unit1.Em4.ControlNodes".cm.brakeTest.cutter.monitoring.error AND NOT #statUnitStatus.acknowledgeActive);
   IF "Unit1.Em4.ControlNodes".cm.brakeTest.cutter.monitoring.error THEN
       "Unit1.Em4.ControlNodes".cm.brakeTest.cutter.monitoring.busy := FALSE;
       "Unit1.Em4.ControlNodes".cm.brakeTest.cutter.commands.axisReset := FALSE;
   END_IF;
   #_w1 := "Unit1.Em4.ControlNodes".cm.brakeTest.cutter.monitoring.busy AND NOT #statPulse[74];   // rising edge
   #statPulse[74] := "Unit1.Em4.ControlNodes".cm.brakeTest.cutter.monitoring.busy;
   IF #_w1 THEN "Unit1.Em4.Config".cmElectrodeCutterAxisZ.disableAlarms := TRUE; END_IF;
   #_w2 := NOT "Unit1.Em4.ControlNodes".cm.brakeTest.cutter.monitoring.busy AND NOT #statPulse[75];   // rising edge
   #statPulse[75] := NOT "Unit1.Em4.ControlNodes".cm.brakeTest.cutter.monitoring.busy;
   IF #_w2 THEN "Unit1.Em4.Config".cmElectrodeCutterAxisZ.disableAlarms := FALSE; END_IF;
END_REGION

REGION Network 116: Cutter Z-Axis Brake Test Initialize
   RUNG wire#powerrail
      { S7_Templates := "SrcType := Int" } GE_Contact(in1 := "Unit1.Em4.ControlNodes".cm.brakeTest.cutter.monitoring."step", in2 := 10)
      { S7_Templates := "SrcType := Int" } LE_Contact(in1 := "Unit1.Em4.ControlNodes".cm.brakeTest.cutter.monitoring."step", in2 := 30)
      P_Contact(operand := #statUnitStatus.mode.production, bit := #statPulse[64])
      wire#w1
      R_Coil( "Unit1.Em4.ControlNodes".cm.brakeTest.cutter.monitoring.busy )
      R_Coil( "Unit1.Em4.ControlNodes".cm.brakeTest.cutter.monitoring.complete )
      R_Coil( "Unit1.Em4.ControlNodes".cm.brakeTest.cutter.commands.axisReset )
   END_RUNG
   RUNG wire#powerrail
      P_Contact(operand := "Unit1.Em4.ControlNodes".cm.brakeTest.cutter.monitoring.error, bit := #statPulse[65])
   END_RUNG wire#w1
   RUNG wire#powerrail
      Contact( "Unit1.Em4.ControlNodes".cm.brakeTest.cutter.monitoring.error )
      wire#w2
      { S7_Templates := "SrcType := Int" } EQ_Contact(in1 := "Unit1.Em4.ControlNodes".cm.brakeTest.cutter.monitoring."step", in2 := 5)
   END_RUNG wire#w1
   RUNG wire#w2
      { S7_Templates := "SrcType := Int" } EQ_Contact(in1 := "Unit1.Em4.ControlNodes".cm.brakeTest.cutter.monitoring."step", in2 := 10)
   END_RUNG wire#w1
   RUNG wire#w1
      Move(in := 0, out1 => "Unit1.Em4.ControlNodes".cm.brakeTest.cutter.monitoring."step")
   END_RUNG
   // the same network as SCL:
   #_w1 := ("Unit1.Em4.ControlNodes".cm.brakeTest.cutter.monitoring."step" >= 10) AND ("Unit1.Em4.ControlNodes".cm.brakeTest.cutter.monitoring."step" <= 30) AND #statUnitStatus.mode.production AND NOT #statPulse[64];   // rising edge of #statUnitStatus.mode.production
   #statPulse[64] := #statUnitStatus.mode.production;
   #_w2 := "Unit1.Em4.ControlNodes".cm.brakeTest.cutter.monitoring.error AND NOT #statPulse[65];   // rising edge of "Unit1.Em4.ControlNodes".cm.brakeTest.cutter.monitoring.error
   #statPulse[65] := "Unit1.Em4.ControlNodes".cm.brakeTest.cutter.monitoring.error;
   IF #_w1 OR #_w2 OR ("Unit1.Em4.ControlNodes".cm.brakeTest.cutter.monitoring.error AND (("Unit1.Em4.ControlNodes".cm.brakeTest.cutter.monitoring."step" = 5) OR ("Unit1.Em4.ControlNodes".cm.brakeTest.cutter.monitoring."step" = 10))) THEN
       "Unit1.Em4.ControlNodes".cm.brakeTest.cutter.monitoring.busy := FALSE;
       "Unit1.Em4.ControlNodes".cm.brakeTest.cutter.monitoring.complete := FALSE;
       "Unit1.Em4.ControlNodes".cm.brakeTest.cutter.commands.axisReset := FALSE;
       "Unit1.Em4.ControlNodes".cm.brakeTest.cutter.monitoring."step" := 0;
   END_IF;
END_REGION

REGION Network 117: Cutter Z-Axis Brake Test Ready
   RUNG wire#powerrail
      Contact( "Unit1.Em4.ControlNodes".cmElectrodeCutterAxisZ.monitoring.axisEnabled )
      Contact( #instLDrv701ControlElectrodeCutterAxisZ.enable )
      Contact( #instLDrv701StatusElectrodeCutterAxisZ.enable )
      Coil( "Unit1.Em4.ControlNodes".cm.brakeTest.cutter.monitoring.ready )
   END_RUNG
   RUNG wire#powerrail
      I_Contact( #instLDrv701ControlElectrodeCutterAxisZ.error )
      Coil( #instLDrv701ControlElectrodeCutterAxisZ.enable )
   END_RUNG
   RUNG wire#powerrail
      I_Contact( #instLDrv701StatusElectrodeCutterAxisZ.error )
      Coil( #instLDrv701StatusElectrodeCutterAxisZ.enable )
   END_RUNG
   // the same network as SCL:
   "Unit1.Em4.ControlNodes".cm.brakeTest.cutter.monitoring.ready := "Unit1.Em4.ControlNodes".cmElectrodeCutterAxisZ.monitoring.axisEnabled AND #instLDrv701ControlElectrodeCutterAxisZ.enable AND #instLDrv701StatusElectrodeCutterAxisZ.enable;
   #instLDrv701ControlElectrodeCutterAxisZ.enable := NOT #instLDrv701ControlElectrodeCutterAxisZ.error;
   #instLDrv701StatusElectrodeCutterAxisZ.enable := NOT #instLDrv701StatusElectrodeCutterAxisZ.error;
END_REGION

REGION Network 118: Cutter Z-Axis Reset
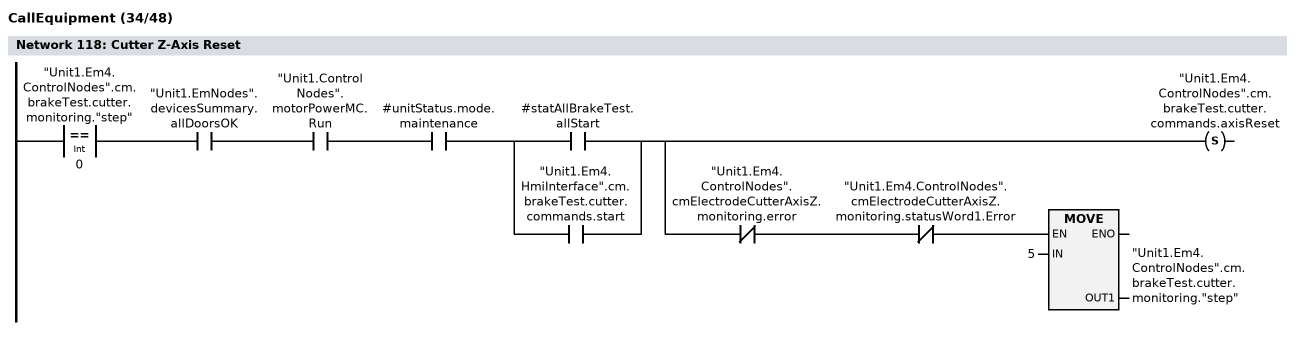
   RUNG wire#powerrail
      { S7_Templates := "SrcType := Int" } EQ_Contact(in1 := "Unit1.Em4.ControlNodes".cm.brakeTest.cutter.monitoring."step", in2 := 0)
      Contact( "Unit1.EmNodes".devicesSummary.allDoorsOK )
      Contact( "Unit1.ControlNodes".motorPowerMC.Run )
      Contact( #unitStatus.mode.maintenance )
      wire#w1
      Contact( #statAllBrakeTest.allStart )
      wire#w2
      S_Coil( "Unit1.Em4.ControlNodes".cm.brakeTest.cutter.commands.axisReset )
   END_RUNG
   RUNG wire#w1
      Contact( "Unit1.Em4.HmiInterface".cm.brakeTest.cutter.commands.start )
   END_RUNG wire#w2
   RUNG wire#w2
      I_Contact( "Unit1.Em4.ControlNodes".cmElectrodeCutterAxisZ.monitoring.error )
      I_Contact( "Unit1.Em4.ControlNodes".cmElectrodeCutterAxisZ.monitoring.statusWord1.Error )
      Move(in := 5, out1 => "Unit1.Em4.ControlNodes".cm.brakeTest.cutter.monitoring."step")
   END_RUNG
   // the same network as SCL:
   #_w1 := ("Unit1.Em4.ControlNodes".cm.brakeTest.cutter.monitoring."step" = 0) AND "Unit1.EmNodes".devicesSummary.allDoorsOK AND "Unit1.ControlNodes".motorPowerMC.Run AND #unitStatus.mode.maintenance AND (#statAllBrakeTest.allStart OR "Unit1.Em4.HmiInterface".cm.brakeTest.cutter.commands.start);
   IF #_w1 THEN "Unit1.Em4.ControlNodes".cm.brakeTest.cutter.commands.axisReset := TRUE; END_IF;
   IF #_w1 AND NOT "Unit1.Em4.ControlNodes".cmElectrodeCutterAxisZ.monitoring.error AND NOT "Unit1.Em4.ControlNodes".cmElectrodeCutterAxisZ.monitoring.statusWord1.Error THEN
       "Unit1.Em4.ControlNodes".cm.brakeTest.cutter.monitoring."step" := 5;
   END_IF;
END_REGION

REGION Network 119: Cutter Z-Axis Brake Test Commands
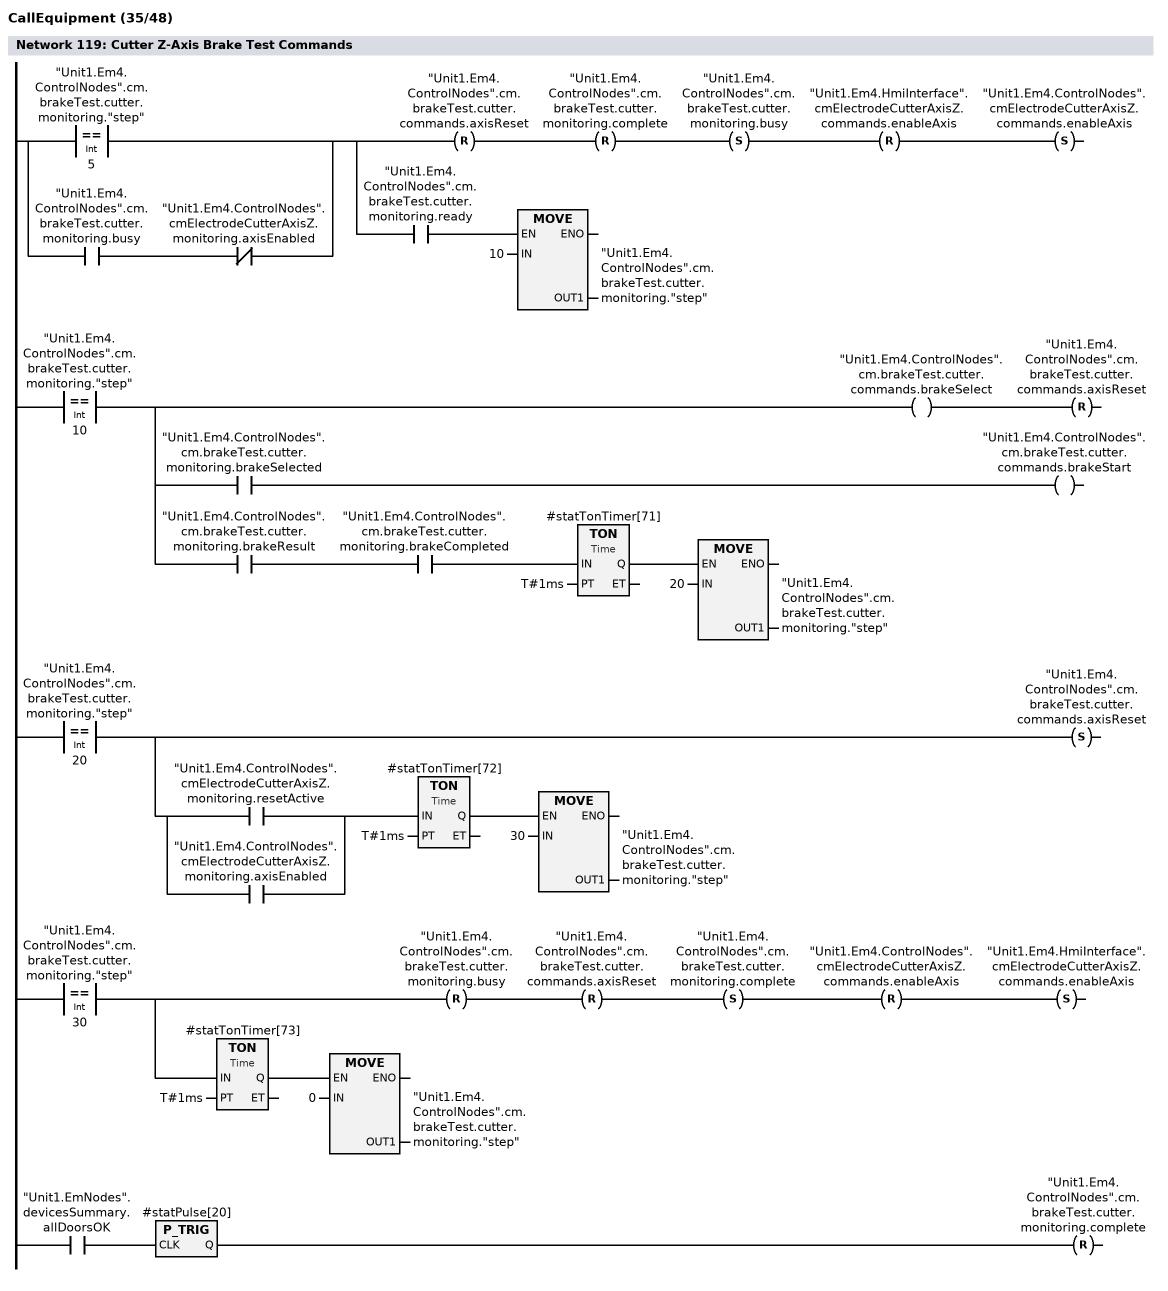
   RUNG wire#powerrail
      { S7_Templates := "SrcType := Int" } EQ_Contact(in1 := "Unit1.Em4.ControlNodes".cm.brakeTest.cutter.monitoring."step", in2 := 5)
      wire#w1
      R_Coil( "Unit1.Em4.ControlNodes".cm.brakeTest.cutter.commands.axisReset )
      R_Coil( "Unit1.Em4.ControlNodes".cm.brakeTest.cutter.monitoring.complete )
      S_Coil( "Unit1.Em4.ControlNodes".cm.brakeTest.cutter.monitoring.busy )
      R_Coil( "Unit1.Em4.HmiInterface".cmElectrodeCutterAxisZ.commands.enableAxis )
      S_Coil( "Unit1.Em4.ControlNodes".cmElectrodeCutterAxisZ.commands.enableAxis )
   END_RUNG
   RUNG wire#powerrail
      Contact( "Unit1.Em4.ControlNodes".cm.brakeTest.cutter.monitoring.busy )
      I_Contact( "Unit1.Em4.ControlNodes".cmElectrodeCutterAxisZ.monitoring.axisEnabled )
   END_RUNG wire#w1
   RUNG wire#w1
      Contact( "Unit1.Em4.ControlNodes".cm.brakeTest.cutter.monitoring.ready )
      Move(in := 10, out1 => "Unit1.Em4.ControlNodes".cm.brakeTest.cutter.monitoring."step")
   END_RUNG
   RUNG wire#powerrail
      { S7_Templates := "SrcType := Int" } EQ_Contact(in1 := "Unit1.Em4.ControlNodes".cm.brakeTest.cutter.monitoring."step", in2 := 10)
      wire#w2
      Coil( "Unit1.Em4.ControlNodes".cm.brakeTest.cutter.commands.brakeSelect )
      R_Coil( "Unit1.Em4.ControlNodes".cm.brakeTest.cutter.commands.axisReset )
   END_RUNG
   RUNG wire#w2
      Contact( "Unit1.Em4.ControlNodes".cm.brakeTest.cutter.monitoring.brakeSelected )
      Coil( "Unit1.Em4.ControlNodes".cm.brakeTest.cutter.commands.brakeStart )
   END_RUNG
   RUNG wire#w2
      Contact( "Unit1.Em4.ControlNodes".cm.brakeTest.cutter.monitoring.brakeResult )
      Contact( "Unit1.Em4.ControlNodes".cm.brakeTest.cutter.monitoring.brakeCompleted )
      { S7_Templates := "time_type := Time" } #statTonTimer[71].TON(pt := T#1ms, et =>)
      Move(in := 20, out1 => "Unit1.Em4.ControlNodes".cm.brakeTest.cutter.monitoring."step")
   END_RUNG
   RUNG wire#powerrail
      { S7_Templates := "SrcType := Int" } EQ_Contact(in1 := "Unit1.Em4.ControlNodes".cm.brakeTest.cutter.monitoring."step", in2 := 20)
      wire#w3
      S_Coil( "Unit1.Em4.ControlNodes".cm.brakeTest.cutter.commands.axisReset )
   END_RUNG
   RUNG wire#w3
      Contact( "Unit1.Em4.ControlNodes".cmElectrodeCutterAxisZ.monitoring.resetActive )
      wire#w4
      { S7_Templates := "time_type := Time" } #statTonTimer[72].TON(pt := T#1ms, et =>)
      Move(in := 30, out1 => "Unit1.Em4.ControlNodes".cm.brakeTest.cutter.monitoring."step")
   END_RUNG
   RUNG wire#w3
      Contact( "Unit1.Em4.ControlNodes".cmElectrodeCutterAxisZ.monitoring.axisEnabled )
   END_RUNG wire#w4
   RUNG wire#powerrail
      { S7_Templates := "SrcType := Int" } EQ_Contact(in1 := "Unit1.Em4.ControlNodes".cm.brakeTest.cutter.monitoring."step", in2 := 30)
      wire#w5
      R_Coil( "Unit1.Em4.ControlNodes".cm.brakeTest.cutter.monitoring.busy )
      R_Coil( "Unit1.Em4.ControlNodes".cm.brakeTest.cutter.commands.axisReset )
      S_Coil( "Unit1.Em4.ControlNodes".cm.brakeTest.cutter.monitoring.complete )
      R_Coil( "Unit1.Em4.ControlNodes".cmElectrodeCutterAxisZ.commands.enableAxis )
      S_Coil( "Unit1.Em4.HmiInterface".cmElectrodeCutterAxisZ.commands.enableAxis )
   END_RUNG
   RUNG wire#w5
      { S7_Templates := "time_type := Time" } #statTonTimer[73].TON(pt := T#1ms, et =>)
      Move(in := 0, out1 => "Unit1.Em4.ControlNodes".cm.brakeTest.cutter.monitoring."step")
   END_RUNG
   RUNG wire#powerrail
      Contact( "Unit1.EmNodes".devicesSummary.allDoorsOK )
      P_Trig( #statPulse[20] )
      R_Coil( "Unit1.Em4.ControlNodes".cm.brakeTest.cutter.monitoring.complete )
   END_RUNG
   // the same network as SCL:
   #_w1 := ("Unit1.Em4.ControlNodes".cm.brakeTest.cutter.monitoring."step" = 5) OR ("Unit1.Em4.ControlNodes".cm.brakeTest.cutter.monitoring.busy AND NOT "Unit1.Em4.ControlNodes".cmElectrodeCutterAxisZ.monitoring.axisEnabled);
   IF #_w1 THEN
       "Unit1.Em4.ControlNodes".cm.brakeTest.cutter.commands.axisReset := FALSE;
       "Unit1.Em4.ControlNodes".cm.brakeTest.cutter.monitoring.complete := FALSE;
       "Unit1.Em4.ControlNodes".cm.brakeTest.cutter.monitoring.busy := TRUE;
       "Unit1.Em4.HmiInterface".cmElectrodeCutterAxisZ.commands.enableAxis := FALSE;
       "Unit1.Em4.ControlNodes".cmElectrodeCutterAxisZ.commands.enableAxis := TRUE;
   END_IF;
   IF #_w1 AND "Unit1.Em4.ControlNodes".cm.brakeTest.cutter.monitoring.ready THEN
       "Unit1.Em4.ControlNodes".cm.brakeTest.cutter.monitoring."step" := 10;
   END_IF;
   "Unit1.Em4.ControlNodes".cm.brakeTest.cutter.commands.brakeSelect := "Unit1.Em4.ControlNodes".cm.brakeTest.cutter.monitoring."step" = 10;
   IF "Unit1.Em4.ControlNodes".cm.brakeTest.cutter.commands.brakeSelect THEN
       "Unit1.Em4.ControlNodes".cm.brakeTest.cutter.commands.axisReset := FALSE;
   END_IF;
   "Unit1.Em4.ControlNodes".cm.brakeTest.cutter.commands.brakeStart := "Unit1.Em4.ControlNodes".cm.brakeTest.cutter.commands.brakeSelect AND "Unit1.Em4.ControlNodes".cm.brakeTest.cutter.monitoring.brakeSelected;
   #statTonTimer[71].TON(IN := "Unit1.Em4.ControlNodes".cm.brakeTest.cutter.commands.brakeSelect AND "Unit1.Em4.ControlNodes".cm.brakeTest.cutter.monitoring.brakeResult AND "Unit1.Em4.ControlNodes".cm.brakeTest.cutter.monitoring.brakeCompleted,
                         PT := T#1ms);
   IF #statTonTimer[71].Q THEN "Unit1.Em4.ControlNodes".cm.brakeTest.cutter.monitoring."step" := 20; END_IF;
   #_w2 := "Unit1.Em4.ControlNodes".cm.brakeTest.cutter.monitoring."step" = 20;
   IF #_w2 THEN "Unit1.Em4.ControlNodes".cm.brakeTest.cutter.commands.axisReset := TRUE; END_IF;
   #statTonTimer[72].TON(IN := #_w2 AND ("Unit1.Em4.ControlNodes".cmElectrodeCutterAxisZ.monitoring.resetActive OR "Unit1.Em4.ControlNodes".cmElectrodeCutterAxisZ.monitoring.axisEnabled),
                         PT := T#1ms);
   IF #statTonTimer[72].Q THEN "Unit1.Em4.ControlNodes".cm.brakeTest.cutter.monitoring."step" := 30; END_IF;
   #_w3 := "Unit1.Em4.ControlNodes".cm.brakeTest.cutter.monitoring."step" = 30;
   IF #_w3 THEN
       "Unit1.Em4.ControlNodes".cm.brakeTest.cutter.monitoring.busy := FALSE;
       "Unit1.Em4.ControlNodes".cm.brakeTest.cutter.commands.axisReset := FALSE;
       "Unit1.Em4.ControlNodes".cm.brakeTest.cutter.monitoring.complete := TRUE;
       "Unit1.Em4.ControlNodes".cmElectrodeCutterAxisZ.commands.enableAxis := FALSE;
       "Unit1.Em4.HmiInterface".cmElectrodeCutterAxisZ.commands.enableAxis := TRUE;
   END_IF;
   #statTonTimer[73].TON(IN := #_w3, PT := T#1ms);
   IF #statTonTimer[73].Q THEN "Unit1.Em4.ControlNodes".cm.brakeTest.cutter.monitoring."step" := 0; END_IF;
   #_w4 := "Unit1.EmNodes".devicesSummary.allDoorsOK AND NOT #statPulse[20];   // rising edge
   #statPulse[20] := "Unit1.EmNodes".devicesSummary.allDoorsOK;
   IF #_w4 THEN "Unit1.Em4.ControlNodes".cm.brakeTest.cutter.monitoring.complete := FALSE; END_IF;
END_REGION

REGION Network 120: Cutter Z-Axis Brake Test Monitoring
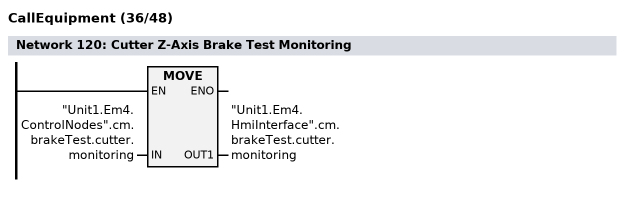
   RUNG wire#powerrail
      Move(in := "Unit1.Em4.ControlNodes".cm.brakeTest.cutter.monitoring, out1 => "Unit1.Em4.HmiInterface".cm.brakeTest.cutter.monitoring)
   END_RUNG
   // the same network as SCL:
   "Unit1.Em4.HmiInterface".cm.brakeTest.cutter.monitoring := "Unit1.Em4.ControlNodes".cm.brakeTest.cutter.monitoring;
END_REGION

REGION Network 121: Call Cutter Z-Axis Telegram 701
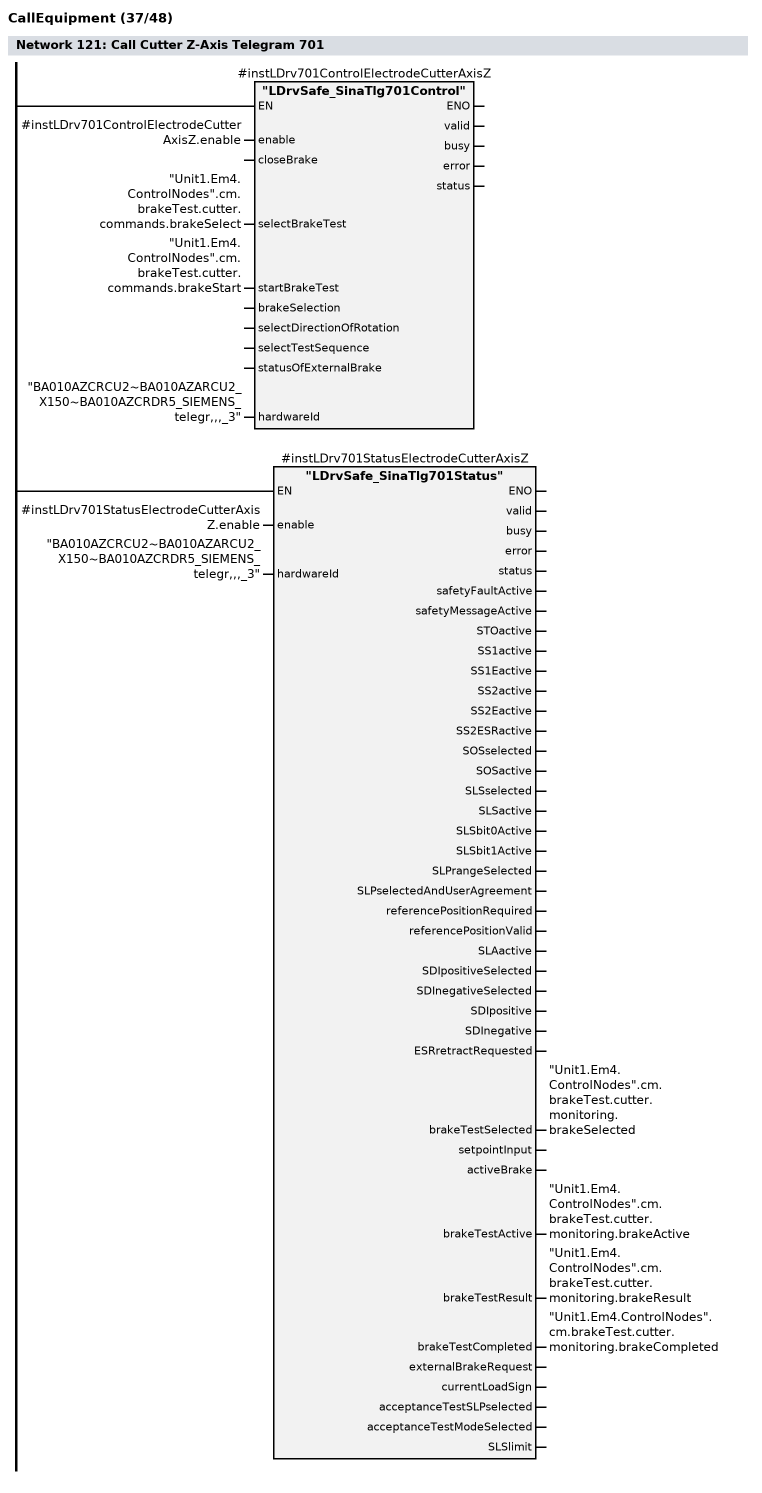
   RUNG wire#powerrail
      #instLDrv701ControlElectrodeCutterAxisZ(enable := #instLDrv701ControlElectrodeCutterAxisZ.enable, closeBrake :=, selectBrakeTest := "Unit1.Em4.ControlNodes".cm.brakeTest.cutter.commands.brakeSelect, startBrakeTest := "Unit1.Em4.ControlNodes".cm.brakeTest.cutter.commands.brakeStart, brakeSelection :=, selectDirectionOfRotation :=, selectTestSequence :=, statusOfExternalBrake :=, hardwareId := "BA010AZCRCU2~BA010AZARCU2_X150~BA010AZCRDR5_SIEMENS_telegr,,,_3", valid =>, busy =>, error =>, status =>)
   END_RUNG
   RUNG wire#powerrail
      #instLDrv701StatusElectrodeCutterAxisZ(enable := #instLDrv701StatusElectrodeCutterAxisZ.enable, hardwareId := "BA010AZCRCU2~BA010AZARCU2_X150~BA010AZCRDR5_SIEMENS_telegr,,,_3", valid =>, busy =>, error =>, status =>, safetyFaultActive =>, safetyMessageActive =>, STOactive =>, SS1active =>, SS1Eactive =>, SS2active =>, SS2Eactive =>, SS2ESRactive =>, SOSselected =>, SOSactive =>, SLSselected =>, SLSactive =>, SLSbit0Active =>, SLSbit1Active =>, SLPrangeSelected =>, SLPselectedAndUserAgreement =>, referencePositionRequired =>, referencePositionValid =>, SLAactive =>, SDIpositiveSelected =>, SDInegativeSelected =>, SDIpositive =>, SDInegative =>, ESRretractRequested =>, brakeTestSelected => "Unit1.Em4.ControlNodes".cm.brakeTest.cutter.monitoring.brakeSelected, setpointInput =>, activeBrake =>, brakeTestActive => "Unit1.Em4.ControlNodes".cm.brakeTest.cutter.monitoring.brakeActive, brakeTestResult => "Unit1.Em4.ControlNodes".cm.brakeTest.cutter.monitoring.brakeResult, brakeTestCompleted => "Unit1.Em4.ControlNodes".cm.brakeTest.cutter.monitoring.brakeCompleted, externalBrakeRequest =>, currentLoadSign =>, acceptanceTestSLPselected =>, acceptanceTestModeSelected =>, SLSlimit =>)
   END_RUNG
   // the same network as SCL:
   #instLDrv701ControlElectrodeCutterAxisZ(enable := #instLDrv701ControlElectrodeCutterAxisZ.enable,   // "LDrvSafe_SinaTlg701Control"
                           selectBrakeTest := "Unit1.Em4.ControlNodes".cm.brakeTest.cutter.commands.brakeSelect,
                           startBrakeTest := "Unit1.Em4.ControlNodes".cm.brakeTest.cutter.commands.brakeStart,
                           hardwareId := "BA010AZCRCU2~BA010AZARCU2_X150~BA010AZCRDR5_SIEMENS_telegr,,,_3");
   #instLDrv701StatusElectrodeCutterAxisZ(enable := #instLDrv701StatusElectrodeCutterAxisZ.enable,   // "LDrvSafe_SinaTlg701Status"
                           hardwareId := "BA010AZCRCU2~BA010AZARCU2_X150~BA010AZCRDR5_SIEMENS_telegr,,,_3",
                           brakeTestSelected => "Unit1.Em4.ControlNodes".cm.brakeTest.cutter.monitoring.brakeSelected,
                           brakeTestActive => "Unit1.Em4.ControlNodes".cm.brakeTest.cutter.monitoring.brakeActive,
                           brakeTestResult => "Unit1.Em4.ControlNodes".cm.brakeTest.cutter.monitoring.brakeResult,
                           brakeTestCompleted => "Unit1.Em4.ControlNodes".cm.brakeTest.cutter.monitoring.brakeCompleted);
END_REGION

REGION Network 123: PositionMoving X-Axis Brake Test Error
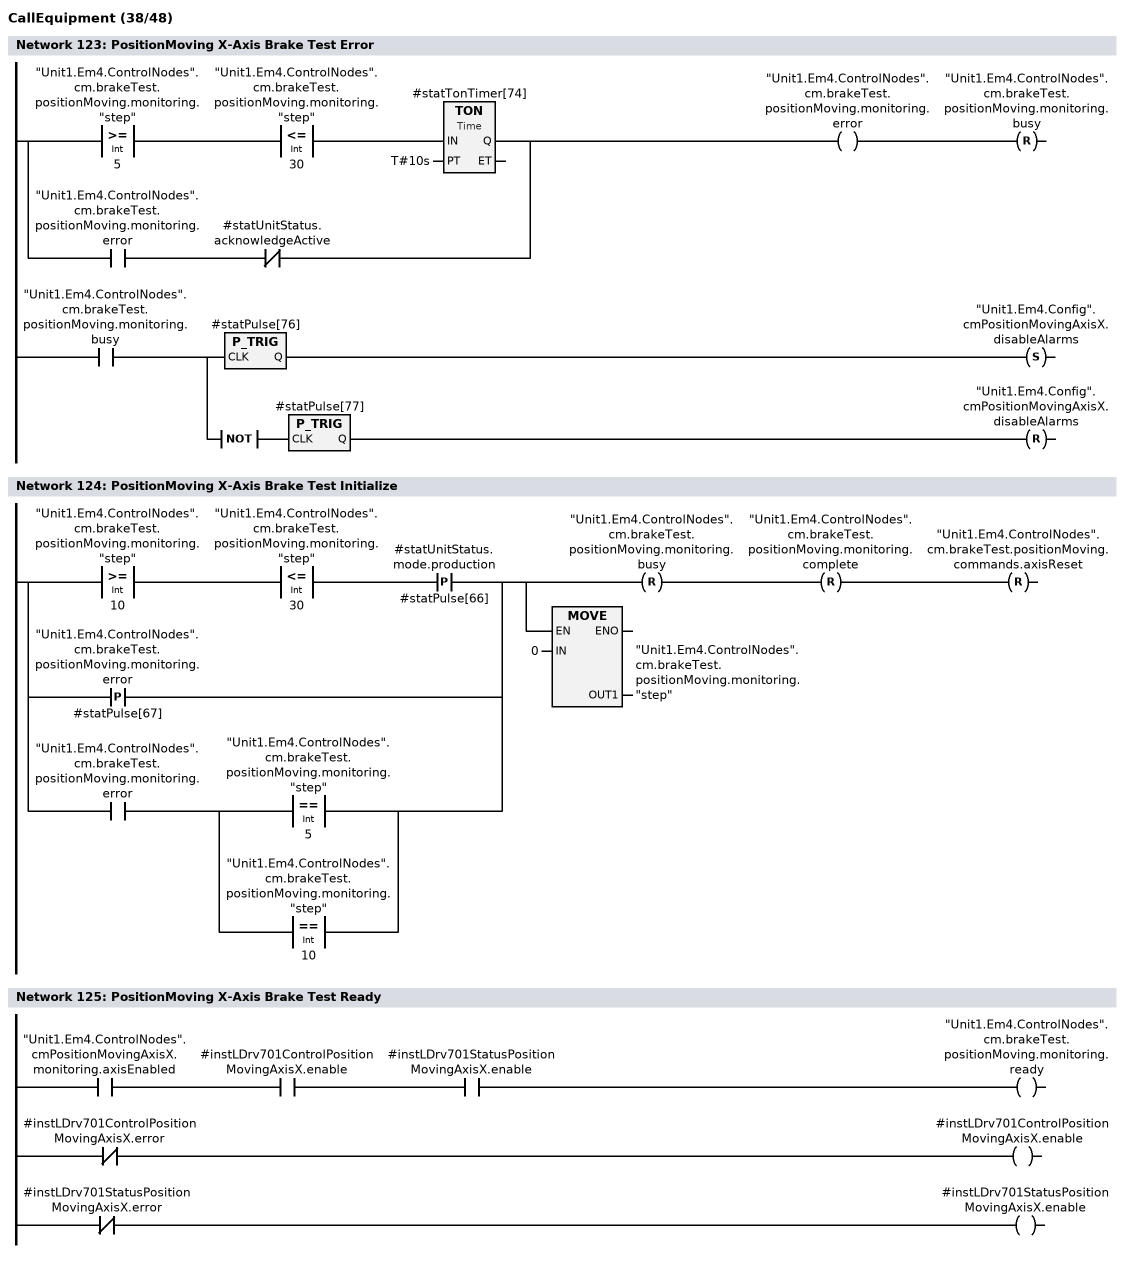
   RUNG wire#powerrail
      { S7_Templates := "SrcType := Int" } GE_Contact(in1 := "Unit1.Em4.ControlNodes".cm.brakeTest.positionMoving.monitoring."step", in2 := 5)
      { S7_Templates := "SrcType := Int" } LE_Contact(in1 := "Unit1.Em4.ControlNodes".cm.brakeTest.positionMoving.monitoring."step", in2 := 30)
      { S7_Templates := "time_type := Time" } #statTonTimer[74].TON(pt := T#10s, et =>)
      wire#w1
      Coil( "Unit1.Em4.ControlNodes".cm.brakeTest.positionMoving.monitoring.error )
      R_Coil( "Unit1.Em4.ControlNodes".cm.brakeTest.positionMoving.monitoring.busy )
   END_RUNG
   RUNG wire#powerrail
      Contact( "Unit1.Em4.ControlNodes".cm.brakeTest.positionMoving.monitoring.error )
      I_Contact( #statUnitStatus.acknowledgeActive )
   END_RUNG wire#w1
   RUNG wire#powerrail
      Contact( "Unit1.Em4.ControlNodes".cm.brakeTest.positionMoving.monitoring.busy )
      wire#w2
      P_Trig( #statPulse[76] )
      S_Coil( "Unit1.Em4.Config".cmPositionMovingAxisX.disableAlarms )
   END_RUNG
   RUNG wire#w2
      Not()
      P_Trig( #statPulse[77] )
      R_Coil( "Unit1.Em4.Config".cmPositionMovingAxisX.disableAlarms )
   END_RUNG
   // the same network as SCL:
   #statTonTimer[74].TON(IN := ("Unit1.Em4.ControlNodes".cm.brakeTest.positionMoving.monitoring."step" >= 5) AND ("Unit1.Em4.ControlNodes".cm.brakeTest.positionMoving.monitoring."step" <= 30),
                         PT := T#10s);
   "Unit1.Em4.ControlNodes".cm.brakeTest.positionMoving.monitoring.error := #statTonTimer[74].Q OR ("Unit1.Em4.ControlNodes".cm.brakeTest.positionMoving.monitoring.error AND NOT #statUnitStatus.acknowledgeActive);
   IF "Unit1.Em4.ControlNodes".cm.brakeTest.positionMoving.monitoring.error THEN
       "Unit1.Em4.ControlNodes".cm.brakeTest.positionMoving.monitoring.busy := FALSE;
   END_IF;
   #_w1 := "Unit1.Em4.ControlNodes".cm.brakeTest.positionMoving.monitoring.busy AND NOT #statPulse[76];   // rising edge
   #statPulse[76] := "Unit1.Em4.ControlNodes".cm.brakeTest.positionMoving.monitoring.busy;
   IF #_w1 THEN "Unit1.Em4.Config".cmPositionMovingAxisX.disableAlarms := TRUE; END_IF;
   #_w2 := NOT "Unit1.Em4.ControlNodes".cm.brakeTest.positionMoving.monitoring.busy AND NOT #statPulse[77];   // rising edge
   #statPulse[77] := NOT "Unit1.Em4.ControlNodes".cm.brakeTest.positionMoving.monitoring.busy;
   IF #_w2 THEN "Unit1.Em4.Config".cmPositionMovingAxisX.disableAlarms := FALSE; END_IF;
END_REGION

REGION Network 124: PositionMoving X-Axis Brake Test Initialize
   RUNG wire#powerrail
      { S7_Templates := "SrcType := Int" } GE_Contact(in1 := "Unit1.Em4.ControlNodes".cm.brakeTest.positionMoving.monitoring."step", in2 := 10)
      { S7_Templates := "SrcType := Int" } LE_Contact(in1 := "Unit1.Em4.ControlNodes".cm.brakeTest.positionMoving.monitoring."step", in2 := 30)
      P_Contact(operand := #statUnitStatus.mode.production, bit := #statPulse[66])
      wire#w1
      R_Coil( "Unit1.Em4.ControlNodes".cm.brakeTest.positionMoving.monitoring.busy )
      R_Coil( "Unit1.Em4.ControlNodes".cm.brakeTest.positionMoving.monitoring.complete )
      R_Coil( "Unit1.Em4.ControlNodes".cm.brakeTest.positionMoving.commands.axisReset )
   END_RUNG
   RUNG wire#powerrail
      P_Contact(operand := "Unit1.Em4.ControlNodes".cm.brakeTest.positionMoving.monitoring.error, bit := #statPulse[67])
   END_RUNG wire#w1
   RUNG wire#powerrail
      Contact( "Unit1.Em4.ControlNodes".cm.brakeTest.positionMoving.monitoring.error )
      wire#w2
      { S7_Templates := "SrcType := Int" } EQ_Contact(in1 := "Unit1.Em4.ControlNodes".cm.brakeTest.positionMoving.monitoring."step", in2 := 5)
   END_RUNG wire#w1
   RUNG wire#w2
      { S7_Templates := "SrcType := Int" } EQ_Contact(in1 := "Unit1.Em4.ControlNodes".cm.brakeTest.positionMoving.monitoring."step", in2 := 10)
   END_RUNG wire#w1
   RUNG wire#w1
      Move(in := 0, out1 => "Unit1.Em4.ControlNodes".cm.brakeTest.positionMoving.monitoring."step")
   END_RUNG
   // the same network as SCL:
   #_w1 := ("Unit1.Em4.ControlNodes".cm.brakeTest.positionMoving.monitoring."step" >= 10) AND ("Unit1.Em4.ControlNodes".cm.brakeTest.positionMoving.monitoring."step" <= 30) AND #statUnitStatus.mode.production AND NOT #statPulse[66];   // rising edge of #statUnitStatus.mode.production
   #statPulse[66] := #statUnitStatus.mode.production;
   #_w2 := "Unit1.Em4.ControlNodes".cm.brakeTest.positionMoving.monitoring.error AND NOT #statPulse[67];   // rising edge of "Unit1.Em4.ControlNodes".cm.brakeTest.positionMoving.monitoring.error
   #statPulse[67] := "Unit1.Em4.ControlNodes".cm.brakeTest.positionMoving.monitoring.error;
   IF #_w1 OR #_w2 OR ("Unit1.Em4.ControlNodes".cm.brakeTest.positionMoving.monitoring.error AND (("Unit1.Em4.ControlNodes".cm.brakeTest.positionMoving.monitoring."step" = 5) OR ("Unit1.Em4.ControlNodes".cm.brakeTest.positionMoving.monitoring."step" = 10))) THEN
       "Unit1.Em4.ControlNodes".cm.brakeTest.positionMoving.monitoring.busy := FALSE;
       "Unit1.Em4.ControlNodes".cm.brakeTest.positionMoving.monitoring.complete := FALSE;
       "Unit1.Em4.ControlNodes".cm.brakeTest.positionMoving.commands.axisReset := FALSE;
       "Unit1.Em4.ControlNodes".cm.brakeTest.positionMoving.monitoring."step" := 0;
   END_IF;
END_REGION

REGION Network 125: PositionMoving X-Axis Brake Test Ready
   RUNG wire#powerrail
      Contact( "Unit1.Em4.ControlNodes".cmPositionMovingAxisX.monitoring.axisEnabled )
      Contact( #instLDrv701ControlPositionMovingAxisX.enable )
      Contact( #instLDrv701StatusPositionMovingAxisX.enable )
      Coil( "Unit1.Em4.ControlNodes".cm.brakeTest.positionMoving.monitoring.ready )
   END_RUNG
   RUNG wire#powerrail
      I_Contact( #instLDrv701ControlPositionMovingAxisX.error )
      Coil( #instLDrv701ControlPositionMovingAxisX.enable )
   END_RUNG
   RUNG wire#powerrail
      I_Contact( #instLDrv701StatusPositionMovingAxisX.error )
      Coil( #instLDrv701StatusPositionMovingAxisX.enable )
   END_RUNG
   // the same network as SCL:
   "Unit1.Em4.ControlNodes".cm.brakeTest.positionMoving.monitoring.ready := "Unit1.Em4.ControlNodes".cmPositionMovingAxisX.monitoring.axisEnabled AND #instLDrv701ControlPositionMovingAxisX.enable AND #instLDrv701StatusPositionMovingAxisX.enable;
   #instLDrv701ControlPositionMovingAxisX.enable := NOT #instLDrv701ControlPositionMovingAxisX.error;
   #instLDrv701StatusPositionMovingAxisX.enable := NOT #instLDrv701StatusPositionMovingAxisX.error;
END_REGION

REGION Network 126: PositionMoving X-Axis Reset
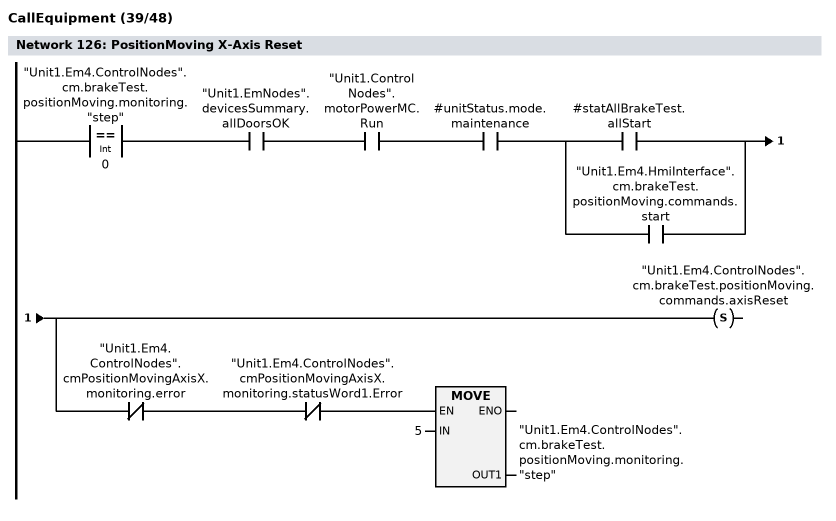
   RUNG wire#powerrail
      { S7_Templates := "SrcType := Int" } EQ_Contact(in1 := "Unit1.Em4.ControlNodes".cm.brakeTest.positionMoving.monitoring."step", in2 := 0)
      Contact( "Unit1.EmNodes".devicesSummary.allDoorsOK )
      Contact( "Unit1.ControlNodes".motorPowerMC.Run )
      Contact( #unitStatus.mode.maintenance )
      wire#w1
      Contact( #statAllBrakeTest.allStart )
      wire#w2
      S_Coil( "Unit1.Em4.ControlNodes".cm.brakeTest.positionMoving.commands.axisReset )
   END_RUNG
   RUNG wire#w1
      Contact( "Unit1.Em4.HmiInterface".cm.brakeTest.positionMoving.commands.start )
   END_RUNG wire#w2
   RUNG wire#w2
      I_Contact( "Unit1.Em4.ControlNodes".cmPositionMovingAxisX.monitoring.error )
      I_Contact( "Unit1.Em4.ControlNodes".cmPositionMovingAxisX.monitoring.statusWord1.Error )
      Move(in := 5, out1 => "Unit1.Em4.ControlNodes".cm.brakeTest.positionMoving.monitoring."step")
   END_RUNG
   // the same network as SCL:
   #_w1 := ("Unit1.Em4.ControlNodes".cm.brakeTest.positionMoving.monitoring."step" = 0) AND "Unit1.EmNodes".devicesSummary.allDoorsOK AND "Unit1.ControlNodes".motorPowerMC.Run AND #unitStatus.mode.maintenance AND (#statAllBrakeTest.allStart OR "Unit1.Em4.HmiInterface".cm.brakeTest.positionMoving.commands.start);
   IF #_w1 THEN "Unit1.Em4.ControlNodes".cm.brakeTest.positionMoving.commands.axisReset := TRUE; END_IF;
   IF #_w1 AND NOT "Unit1.Em4.ControlNodes".cmPositionMovingAxisX.monitoring.error AND NOT "Unit1.Em4.ControlNodes".cmPositionMovingAxisX.monitoring.statusWord1.Error THEN
       "Unit1.Em4.ControlNodes".cm.brakeTest.positionMoving.monitoring."step" := 5;
   END_IF;
END_REGION

REGION Network 127: PositionMoving X-Axis Brake Test Commands
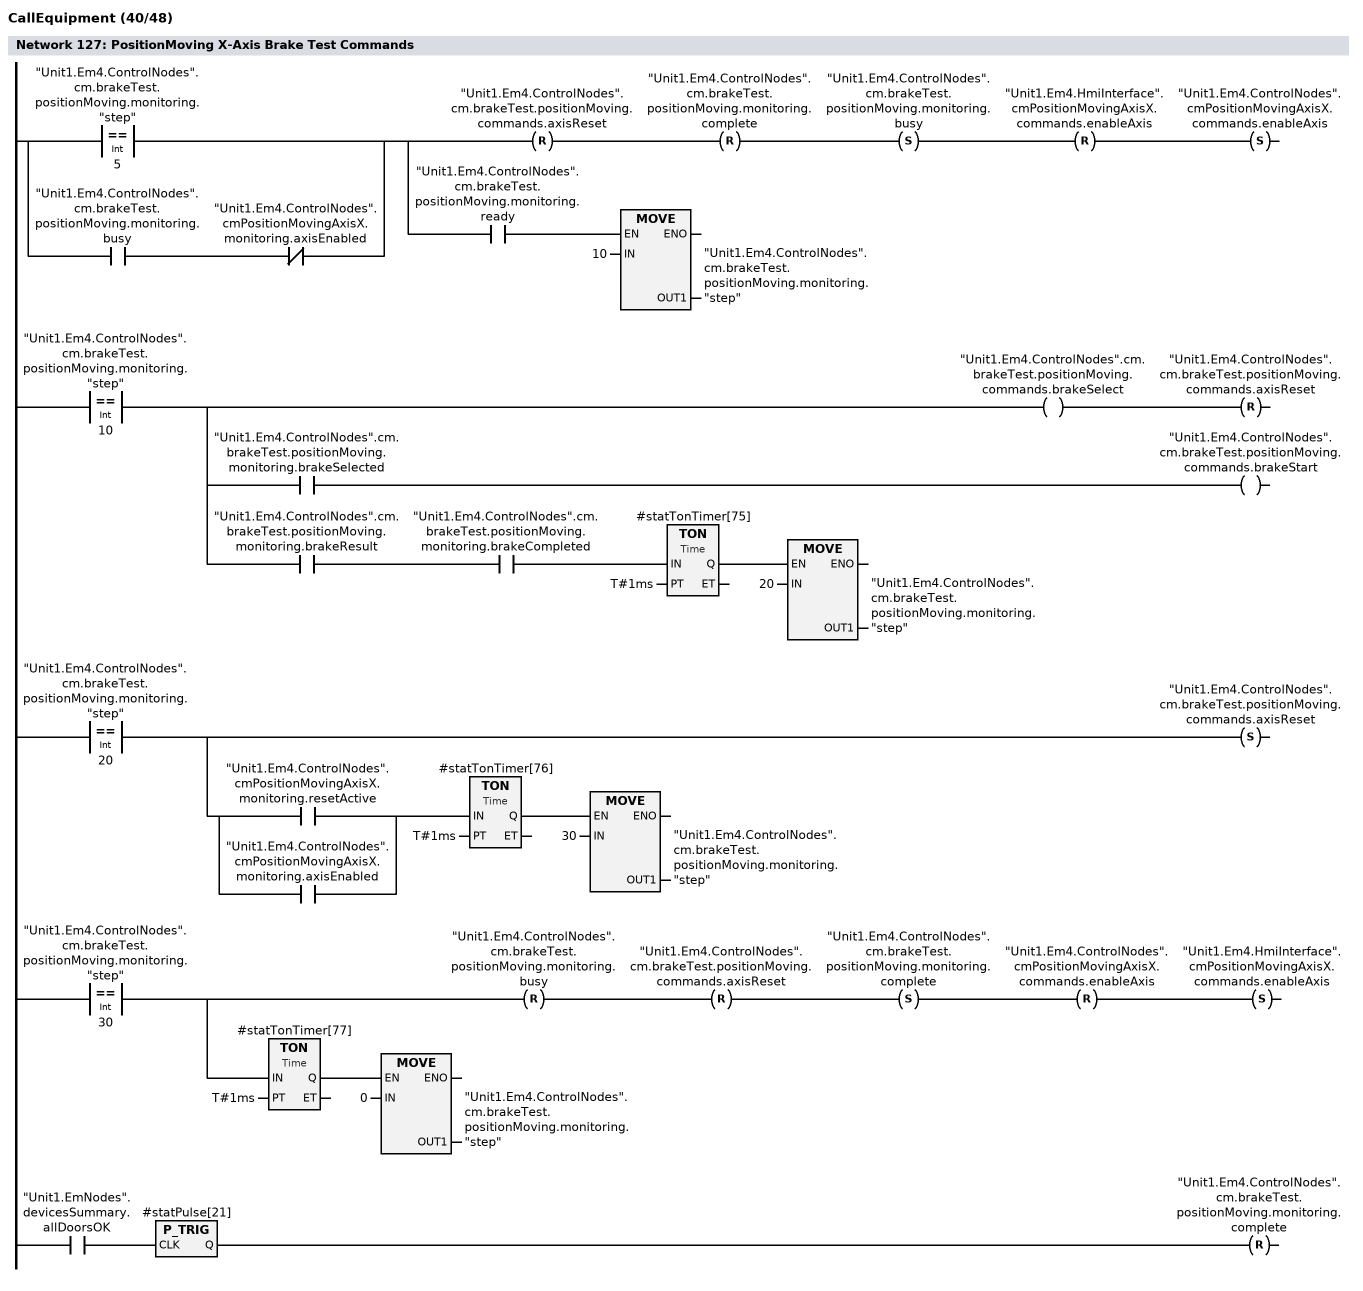
   RUNG wire#powerrail
      { S7_Templates := "SrcType := Int" } EQ_Contact(in1 := "Unit1.Em4.ControlNodes".cm.brakeTest.positionMoving.monitoring."step", in2 := 5)
      wire#w1
      R_Coil( "Unit1.Em4.ControlNodes".cm.brakeTest.positionMoving.commands.axisReset )
      R_Coil( "Unit1.Em4.ControlNodes".cm.brakeTest.positionMoving.monitoring.complete )
      S_Coil( "Unit1.Em4.ControlNodes".cm.brakeTest.positionMoving.monitoring.busy )
      R_Coil( "Unit1.Em4.HmiInterface".cmPositionMovingAxisX.commands.enableAxis )
      S_Coil( "Unit1.Em4.ControlNodes".cmPositionMovingAxisX.commands.enableAxis )
   END_RUNG
   RUNG wire#powerrail
      Contact( "Unit1.Em4.ControlNodes".cm.brakeTest.positionMoving.monitoring.busy )
      I_Contact( "Unit1.Em4.ControlNodes".cmPositionMovingAxisX.monitoring.axisEnabled )
   END_RUNG wire#w1
   RUNG wire#w1
      Contact( "Unit1.Em4.ControlNodes".cm.brakeTest.positionMoving.monitoring.ready )
      Move(in := 10, out1 => "Unit1.Em4.ControlNodes".cm.brakeTest.positionMoving.monitoring."step")
   END_RUNG
   RUNG wire#powerrail
      { S7_Templates := "SrcType := Int" } EQ_Contact(in1 := "Unit1.Em4.ControlNodes".cm.brakeTest.positionMoving.monitoring."step", in2 := 10)
      wire#w2
      Coil( "Unit1.Em4.ControlNodes".cm.brakeTest.positionMoving.commands.brakeSelect )
      R_Coil( "Unit1.Em4.ControlNodes".cm.brakeTest.positionMoving.commands.axisReset )
   END_RUNG
   RUNG wire#w2
      Contact( "Unit1.Em4.ControlNodes".cm.brakeTest.positionMoving.monitoring.brakeSelected )
      Coil( "Unit1.Em4.ControlNodes".cm.brakeTest.positionMoving.commands.brakeStart )
   END_RUNG
   RUNG wire#w2
      Contact( "Unit1.Em4.ControlNodes".cm.brakeTest.positionMoving.monitoring.brakeResult )
      Contact( "Unit1.Em4.ControlNodes".cm.brakeTest.positionMoving.monitoring.brakeCompleted )
      { S7_Templates := "time_type := Time" } #statTonTimer[75].TON(pt := T#1ms, et =>)
      Move(in := 20, out1 => "Unit1.Em4.ControlNodes".cm.brakeTest.positionMoving.monitoring."step")
   END_RUNG
   RUNG wire#powerrail
      { S7_Templates := "SrcType := Int" } EQ_Contact(in1 := "Unit1.Em4.ControlNodes".cm.brakeTest.positionMoving.monitoring."step", in2 := 20)
      wire#w3
      S_Coil( "Unit1.Em4.ControlNodes".cm.brakeTest.positionMoving.commands.axisReset )
   END_RUNG
   RUNG wire#w3
      Contact( "Unit1.Em4.ControlNodes".cmPositionMovingAxisX.monitoring.resetActive )
      wire#w4
      { S7_Templates := "time_type := Time" } #statTonTimer[76].TON(pt := T#1ms, et =>)
      Move(in := 30, out1 => "Unit1.Em4.ControlNodes".cm.brakeTest.positionMoving.monitoring."step")
   END_RUNG
   RUNG wire#w3
      Contact( "Unit1.Em4.ControlNodes".cmPositionMovingAxisX.monitoring.axisEnabled )
   END_RUNG wire#w4
   RUNG wire#powerrail
      { S7_Templates := "SrcType := Int" } EQ_Contact(in1 := "Unit1.Em4.ControlNodes".cm.brakeTest.positionMoving.monitoring."step", in2 := 30)
      wire#w5
      R_Coil( "Unit1.Em4.ControlNodes".cm.brakeTest.positionMoving.monitoring.busy )
      R_Coil( "Unit1.Em4.ControlNodes".cm.brakeTest.positionMoving.commands.axisReset )
      S_Coil( "Unit1.Em4.ControlNodes".cm.brakeTest.positionMoving.monitoring.complete )
      R_Coil( "Unit1.Em4.ControlNodes".cmPositionMovingAxisX.commands.enableAxis )
      S_Coil( "Unit1.Em4.HmiInterface".cmPositionMovingAxisX.commands.enableAxis )
   END_RUNG
   RUNG wire#w5
      { S7_Templates := "time_type := Time" } #statTonTimer[77].TON(pt := T#1ms, et =>)
      Move(in := 0, out1 => "Unit1.Em4.ControlNodes".cm.brakeTest.positionMoving.monitoring."step")
   END_RUNG
   RUNG wire#powerrail
      Contact( "Unit1.EmNodes".devicesSummary.allDoorsOK )
      P_Trig( #statPulse[21] )
      R_Coil( "Unit1.Em4.ControlNodes".cm.brakeTest.positionMoving.monitoring.complete )
   END_RUNG
   // the same network as SCL:
   #_w1 := ("Unit1.Em4.ControlNodes".cm.brakeTest.positionMoving.monitoring."step" = 5) OR ("Unit1.Em4.ControlNodes".cm.brakeTest.positionMoving.monitoring.busy AND NOT "Unit1.Em4.ControlNodes".cmPositionMovingAxisX.monitoring.axisEnabled);
   IF #_w1 THEN
       "Unit1.Em4.ControlNodes".cm.brakeTest.positionMoving.commands.axisReset := FALSE;
       "Unit1.Em4.ControlNodes".cm.brakeTest.positionMoving.monitoring.complete := FALSE;
       "Unit1.Em4.ControlNodes".cm.brakeTest.positionMoving.monitoring.busy := TRUE;
       "Unit1.Em4.HmiInterface".cmPositionMovingAxisX.commands.enableAxis := FALSE;
       "Unit1.Em4.ControlNodes".cmPositionMovingAxisX.commands.enableAxis := TRUE;
   END_IF;
   IF #_w1 AND "Unit1.Em4.ControlNodes".cm.brakeTest.positionMoving.monitoring.ready THEN
       "Unit1.Em4.ControlNodes".cm.brakeTest.positionMoving.monitoring."step" := 10;
   END_IF;
   "Unit1.Em4.ControlNodes".cm.brakeTest.positionMoving.commands.brakeSelect := "Unit1.Em4.ControlNodes".cm.brakeTest.positionMoving.monitoring."step" = 10;
   IF "Unit1.Em4.ControlNodes".cm.brakeTest.positionMoving.commands.brakeSelect THEN
       "Unit1.Em4.ControlNodes".cm.brakeTest.positionMoving.commands.axisReset := FALSE;
   END_IF;
   "Unit1.Em4.ControlNodes".cm.brakeTest.positionMoving.commands.brakeStart := "Unit1.Em4.ControlNodes".cm.brakeTest.positionMoving.commands.brakeSelect AND "Unit1.Em4.ControlNodes".cm.brakeTest.positionMoving.monitoring.brakeSelected;
   #statTonTimer[75].TON(IN := "Unit1.Em4.ControlNodes".cm.brakeTest.positionMoving.commands.brakeSelect AND "Unit1.Em4.ControlNodes".cm.brakeTest.positionMoving.monitoring.brakeResult AND "Unit1.Em4.ControlNodes".cm.brakeTest.positionMoving.monitoring.brakeCompleted,
                         PT := T#1ms);
   IF #statTonTimer[75].Q THEN
       "Unit1.Em4.ControlNodes".cm.brakeTest.positionMoving.monitoring."step" := 20;
   END_IF;
   #_w2 := "Unit1.Em4.ControlNodes".cm.brakeTest.positionMoving.monitoring."step" = 20;
   IF #_w2 THEN "Unit1.Em4.ControlNodes".cm.brakeTest.positionMoving.commands.axisReset := TRUE; END_IF;
   #statTonTimer[76].TON(IN := #_w2 AND ("Unit1.Em4.ControlNodes".cmPositionMovingAxisX.monitoring.resetActive OR "Unit1.Em4.ControlNodes".cmPositionMovingAxisX.monitoring.axisEnabled),
                         PT := T#1ms);
   IF #statTonTimer[76].Q THEN
       "Unit1.Em4.ControlNodes".cm.brakeTest.positionMoving.monitoring."step" := 30;
   END_IF;
   #_w3 := "Unit1.Em4.ControlNodes".cm.brakeTest.positionMoving.monitoring."step" = 30;
   IF #_w3 THEN
       "Unit1.Em4.ControlNodes".cm.brakeTest.positionMoving.monitoring.busy := FALSE;
       "Unit1.Em4.ControlNodes".cm.brakeTest.positionMoving.commands.axisReset := FALSE;
       "Unit1.Em4.ControlNodes".cm.brakeTest.positionMoving.monitoring.complete := TRUE;
       "Unit1.Em4.ControlNodes".cmPositionMovingAxisX.commands.enableAxis := FALSE;
       "Unit1.Em4.HmiInterface".cmPositionMovingAxisX.commands.enableAxis := TRUE;
   END_IF;
   #statTonTimer[77].TON(IN := #_w3, PT := T#1ms);
   IF #statTonTimer[77].Q THEN
       "Unit1.Em4.ControlNodes".cm.brakeTest.positionMoving.monitoring."step" := 0;
   END_IF;
   #_w4 := "Unit1.EmNodes".devicesSummary.allDoorsOK AND NOT #statPulse[21];   // rising edge
   #statPulse[21] := "Unit1.EmNodes".devicesSummary.allDoorsOK;
   IF #_w4 THEN "Unit1.Em4.ControlNodes".cm.brakeTest.positionMoving.monitoring.complete := FALSE; END_IF;
END_REGION

REGION Network 128: PositionMoving X-Axis Brake Test Monitoring
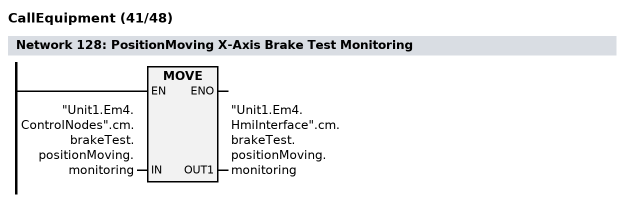
   RUNG wire#powerrail
      Move(in := "Unit1.Em4.ControlNodes".cm.brakeTest.positionMoving.monitoring, out1 => "Unit1.Em4.HmiInterface".cm.brakeTest.positionMoving.monitoring)
   END_RUNG
   // the same network as SCL:
   "Unit1.Em4.HmiInterface".cm.brakeTest.positionMoving.monitoring := "Unit1.Em4.ControlNodes".cm.brakeTest.positionMoving.monitoring;
END_REGION

